// TIA Portal project "Elevador" (V16)

(* hardware
DEVICE "S71500/ET200MP station_1"  S7-1500 station
   slot 0: "Rail_0"  Rack  6ES7 590-1***0-0AA0
   slot 1: "PLC_1"  CPU 1516-3 PN/DP  6ES7 516-3AN00-0AB0  V1.8
      slot 3: "CPU display_1"  6ES7591-1BA00-0AA0
      slot 32768: "PROFINET interface_1"  X1
         slot 32769: "Port_1"  X1 P1
         slot 32770: "Port_2"  X1 P2
      slot 33024: "PROFINET interface_2"  X2
         slot 33025: "Port_1"  X2 P1
      slot 33280: "DP interface_1"  X3
DEVICE "HMI_1"  TP700 Comfort
   slot 0: "HMI_1"  TP700 Comfort  6AV2 124-0GC01-0AX0  16.0.0.0
   slot 1: "HMI_RT_1"  TP700 Comfort  6AV2 124-0GC01-0AX0  16.0.0.0
   slot 5: "HMI_1.IE_CP_1"  PROFINET Interface  16.0.0.0
      slot 1: "PROFINET Interface_1"  PROFINET Interface
         slot 1: "Port_1"  Port
         slot 2: "Port_2"  Port
   slot 7: "HMI_1.MPI/DP_CP_1"  MPI/DP Interface  16.0.0.0
DEVICE "HMI_2"  TP700 Comfort
   slot 0: "HMI_2"  TP700 Comfort  6AV2 124-0GC01-0AX0  16.0.0.0
   slot 1: "HMI_RT_2"  TP700 Comfort  6AV2 124-0GC01-0AX0  16.0.0.0
   slot 5: "HMI_2.IE_CP_1"  PROFINET Interface  16.0.0.0
      slot 1: "PROFINET Interface_1"  PROFINET Interface
         slot 1: "Port_1"  Port
         slot 2: "Port_2"  Port
   slot 7: "HMI_2.MPI/DP_CP_1"  MPI/DP Interface  16.0.0.0
*)

// ===== PLC "PLC_1"  CPU 1516-3 PN/DP =====

VAR_GLOBAL   // PLC tag table "Default tag table"
   "posGround" AT %I0.0 : Bool;   // Sensor Elevador En Planta Baja
   "posFloor1" AT %I0.1 : Bool;   // Sensor Elevador en Primer Piso
   "posFloor2" AT %I0.2 : Bool;   // Sensor Elevador en Segundo Piso
   "posFloor3" AT %I0.3 : Bool;   // Sensor Elevador en Tercer Piso
   "slowGround" AT %I0.4 : Bool;   // Sensor Cambio a Vel Reducida PB
   "slowBottom1" AT %I0.5 : Bool;   // Sensor Cambio Vel Reducida PP Abajo
   "slowTop1" AT %I0.6 : Bool;   // Sensor Cambio Vel Reducida PP Arriba
   "slowBottom2" AT %I0.7 : Bool;   // Sensor Cambio Vel Reducida SP Abajo
   "slowTop2" AT %I1.0 : Bool;   // Sensor Cambio Vel Reducida SP Arriba
   "slow3" AT %I1.1 : Bool;   // Sensor Cambio a Vel Reducida TP
   "doorOpenedG" AT %I1.2 : Bool;   // Sensor Puerta Abierta en Planta Baja
   "doorClosedG" AT %I1.3 : Bool;   // Sensor Puerta Cerrada en Planta Baja
   "doorOpened1" AT %I1.4 : Bool;   // Sensor Puerta Abierta en Primer Piso
   "doorClosed1" AT %I1.5 : Bool;   // Sensor Puerta Cerrada en Primer Piso
   "doorOpened2" AT %I1.6 : Bool;   // Sensor Puerta Abierta en Segundo Piso
   "doorClosed2" AT %I1.7 : Bool;   // Sensor Puerta Cerrada en Segundo Piso
   "doorOpened3" AT %I2.0 : Bool;   // Sensor Puerta Abierta en Tercer Piso
   "doorClosed3" AT %I2.1 : Bool;   // Sensor Puerta Cerrada en Tercer Piso
   "lightBGround" AT %I2.2 : Bool;   // Sensor Luz Puerta en Planta Baja
   "lightB1" AT %I2.3 : Bool;   // Sensor Luz Puerta en Primer Piso
   "lightB2" AT %I2.4 : Bool;   // Sensor Luz Puerta en Segundo Piso
   "lightB3" AT %I2.5 : Bool;   // Sensor Luz Puerta en Tercer Piso
   "sendGround" AT %I4.0 : Bool;   // Boton (NC) para envio a Planta Baja
   "send1" AT %I4.1 : Bool;   // Boton (NC) para envio a Primer Piso
   "send2" AT %I4.2 : Bool;   // Boton (NC) para envio a Segundo Piso
   "send3" AT %I4.3 : Bool;   // Boton (NC) para envio a Tercer Piso
   "alert" AT %I4.4 : Bool;   // Boton (NC) para Alerta
   "emergency" AT %I4.5 : Bool;   // Boton (NC) para Paro Emergencia
   "callGround" AT %I5.0 : Bool;   // Boton (NC) para llamar en Planta Baja
   "callDown1" AT %I5.1 : Bool;   // Boton (NC) para llamar Abajo Primer Piso
   "callUp1" AT %I5.2 : Bool;   // Boton (NC) para llamar Arriba Primer Piso
   "callDown2" AT %I5.3 : Bool;   // Boton (NC) para llamar Abajo Segundo Piso
   "callUp2" AT %I5.4 : Bool;   // Boton (NC) para llamar Arriba Segundo Piso
   "call3" AT %I5.5 : Bool;   // Boton (NC) para llamar en Tercer Piso
   "overload" AT %I5.6 : Bool;   // Boton (NC) de Sobrecarga por Peso
   "toZ+" AT %Q0.0 : Bool;   // Motor Elevador Hacia Arriba
   "toZ-" AT %Q0.1 : Bool;   // Motor Elevador Hacia Abajo
   "slow" AT %Q0.2 : Bool;   // Activar Velocidad Reducida Relevador
   "openDoorG" AT %Q0.3 : Bool;   // Puerta Abrir Planta Baja Piston
   "closeDoorG" AT %Q0.4 : Bool;   // Puerta Cerrar Planta Baja Piston
   "openDoor1" AT %Q0.5 : Bool;   // Puerta Abrir Primer Piso Piston
   "closeDoor1" AT %Q0.6 : Bool;   // Puerta Cerrar Primer Piso Piston
   "openDoor2" AT %Q0.7 : Bool;   // Puerta Abrir Segundo Piso Piston
   "closeDoor2" AT %Q1.0 : Bool;   // Puerta Cerrar Segundo Piso Piston
   "openDoor3" AT %Q1.1 : Bool;   // Puerta Abrir Tercer Piso Piston
   "closeDoor3" AT %Q1.2 : Bool;   // Puerta Cerrar Tercer Piso Piston
   "callToGround" AT %Q1.3 : Bool;   // LED Llamar Planta Baja
   "callToDown1" AT %Q1.4 : Bool;   // LED Llamar Abajo Primer Piso
   "callToUp1" AT %Q1.5 : Bool;   // LED Llamar Arriba Primer Piso
   "callToDown2" AT %Q1.6 : Bool;   // LED Llamar Abajo Segundo Piso
   "callToUp2" AT %Q1.7 : Bool;   // LED Llamar Arriba Segundo Piso
   "callTo3" AT %Q2.0 : Bool;   // LED Llamar Tercer Piso
   "floorIndicatorG" AT %Q2.1 : Bool;   // LED Elevador en Planta Baja
   "floorIndicator1" AT %Q2.2 : Bool;   // LED Elevador en Primer Piso
   "floorIndicator2" AT %Q2.3 : Bool;   // LED Elevador en Segundo Piso
   "floorIndicator3" AT %Q2.4 : Bool;   // LED Elevador en Tercer Piso
   "cabinDown" AT %Q2.5 : Bool;   // LED Elevador Moviendose hacia Abajo
   "cabinUp" AT %Q2.6 : Bool;   // LED Elevador Moviendose hacia Arriba
   "sendToGround" AT %Q2.7 : Bool;   // LED Envio a Planta Baja
   "sendTo1" AT %Q3.0 : Bool;   // LED Envio a Primer Piso
   "sendTo2" AT %Q3.1 : Bool;   // LED Envio a Segundo Piso
   "sendTo3" AT %Q3.2 : Bool;   // LED Envio a Tercer Piso
   "alertInd" AT %Q3.3 : Bool;   // LED Alerta Activada
   "emergencyInd" AT %Q3.4 : Bool;   // LED Paro de Emergencia Activado
   "overloadInd" AT %Q3.5 : Bool;   // LED Sobrecarga Detectada
   "sendGroundMaster" AT %M0.1 : Bool;
   "send1Master" AT %M0.2 : Bool;
   "send2Master" AT %M0.3 : Bool;
   "send3Master" AT %M0.4 : Bool;
   "alertMaster" AT %M0.5 : Bool;
   "emergencyMaster" AT %M0.6 : Bool;
   "abrirPuertasMaster" AT %M0.7 : Bool;
   "cerrarPuertasMaster" AT %M1.0 : Bool;
   "tempFloor1" AT %M1.1 : Bool;
   "tempFloor2" AT %M1.2 : Bool;
   "tempFloor3" AT %M1.3 : Bool;
   "tempFloor4" AT %M1.4 : Bool;
   "tempFloor5" AT %M1.5 : Bool;
   "tempFloor6" AT %M1.6 : Bool;
   "tempFloor7" AT %M1.7 : Bool;
   "sendTo3Master" AT %M2.0 : Bool;
   "sendTo2Master" AT %M2.1 : Bool;
   "sendTo1Master" AT %M2.2 : Bool;
   "sendToGroundMaster" AT %M2.3 : Bool;
   "alertIndMaster" AT %M2.4 : Bool;
   "emergencyIndMaster" AT %M2.5 : Bool;
END_VAR

DATA_BLOCK "Var"   // DB1
{ S7_Optimized_Access := 'TRUE' }
VERSION : 0.1
   VAR
      Acc : Array[0..10] of String;
      AccMovTemp : Array[0..10] of String;
      Ind : Array[0..15] of Bool;
      AccSucc : Array[0..15] of Bool;
      bounceOneAlerta : Bool;
      bounceTwoAlerta : Bool;
      bounceOneEmergen : Bool;
      bounceTwoEmergen : Bool;
      bounceOneGroundA : Bool;
      sendAccGroundA : Bool;
      PuertaIniciada : Bool;
      PuertaAbriendo : Bool;
      PuertaAbierta : Bool;
      PuertaCerrando : Bool;
      PuertaInterrumpida : Bool;
      PuertaTerminada : Bool;
      PuertaTimerInicio : Bool;
      PuertaTimerTermino : Bool;
      PuertaInterrBounce : Bool;
      ActivarPuertaGA : Bool;
      ActivarPuertaF1 : Bool;
      ActivarPuertaF2 : Bool;
      ActivarPuertaF3 : Bool;
      bounceOneF1DownA : Bool;
      sendAccF1DownA : Bool;
      tempStringOne : String;
      tempStringTwo : String;
      ACCION : Bool;
      DeGAaF1 : Bool;
      DeGAaF2 : Bool;
      DeGAaF3 : Bool;
      DeF1aGA : Bool;
      DeF1aF2 : Bool;
      DeF1aF3 : Bool;
      DeF2aGA : Bool;
      DeF2aF1 : Bool;
      DeF2aF3 : Bool;
      DeF3aGA : Bool;
      DeF3aF1 : Bool;
      DeF3aF2 : Bool;
      MOVIMIENTO : Bool;
      MovimientoLento : Bool;
      MovimientoRapido : Bool;
      MASTER : Bool;
      SimuladorEstado1 : Bool;
      SimuladorEstado2 : Bool;
      SimuladorEstado3 : Bool;
      SimuladorEstado4 : Bool;
      SimuladorEstado5 : Bool;
      SimuladorEstado6 : Bool;
      SimuladorEstado7 : Bool;
      SimuladorEstado8 : Bool;
      MASTERINDICATOR : Bool;
      MasterBounceOne : Bool;
      MasterBounceTwo : Bool;
      MasterBounceThree : Bool;
      RESET : Bool;
      ResetApplied : Bool;
      MasterResetPos : Bool;
      MasterResPosPuerta : Bool;
      MasterPuertaG : Bool;
      MasterPuerta1 : Bool;
      MasterPuerta2 : Bool;
      MasterPuerta3 : Bool;
      MasterPuertaGBounce : Bool;
      MasterPuertaGBounce2 : Bool;
      MasterPuerta1Bounce : Bool;
      MasterPuerta1Bounce2 : Bool;
      MasterPuerta2Bounce : Bool;
      MasterPuerta2Bounce2 : Bool;
      MasterPuerta3Bounce : Bool;
      MasterPuerta3Bounce2 : Bool;
      MasterSendToGround : Bool;
      MasterSendTo1 : Bool;
      MasterSendTo2 : Bool;
      MasterSendTo3 : Bool;
      MasterSendToGroundB : Bool;
      MasterSendToGroundB2 : Bool;
      MasterSendTo1B : Bool;
      MasterSendTo1B2 : Bool;
      MasterSendTo2B : Bool;
      MasterSendTo2B2 : Bool;
      MasterSendTo3B : Bool;
      MasterSendTo3B2 : Bool;
      MasterAlertaB1 : Bool;
      MasterAlertaB2 : Bool;
      MasterAlertaB3 : Bool;
      MasterEmergencyB1 : Bool;
      MasterEmergencyB2 : Bool;
      MasterEmergencyB3 : Bool;
      bounceOneF1UpA : Bool;
      sendAccF1UpA : Bool;
      bounceOneF2DownA : Bool;
      sendAccF2DownA : Bool;
      bounceOneF2UpA : Bool;
      sendAccF2UpA : Bool;
      bounceOneF3A : Bool;
      sendAccF3A : Bool;
      bounceGroundPanel : Bool;
      sendAccGroundPanel : Bool;
      bounceF1Panel : Bool;
      sendAccF1Panel : Bool;
      bounceF2Panel : Bool;
      sendAccF2Panel : Bool;
      bounceF3Panel : Bool;
      sendAccF3Panel : Bool;
      bouncePanelF31 : Bool;
      bouncePanelF32 : Bool;
      bouncePanelF33 : Bool;
      bouncePanelF21 : Bool;
      bouncePanelF22 : Bool;
      bouncePanelF23 : Bool;
      bouncePanelF11 : Bool;
      bouncePanelF12 : Bool;
      bouncePanelF13 : Bool;
      bouncePanelFG1 : Bool;
      bouncePanelFG2 : Bool;
      bouncePanelFG3 : Bool;
      Accion2 : Bool;
      Accion3 : Bool;
      TEST : Bool;
      IndTimerInicio : Bool;
      IndTimerTermino : Bool;
      Ultimo : String;
      LimpiarUltimo : Bool;
   END_VAR
BEGIN
   Acc[0] := 'EMPTY';
   Acc[1] := 'EMPTY';
   Acc[2] := 'EMPTY';
   Acc[3] := 'EMPTY';
   Acc[4] := 'EMPTY';
   Acc[5] := 'EMPTY';
   Acc[6] := 'EMPTY';
   Acc[7] := 'EMPTY';
   Acc[8] := 'EMPTY';
   Acc[9] := 'EMPTY';
   Acc[10] := 'EMPTY';
   AccMovTemp[0] := 'EMPTY';
   AccMovTemp[1] := 'EMPTY';
   AccMovTemp[2] := 'EMPTY';
   AccMovTemp[3] := 'EMPTY';
   AccMovTemp[4] := 'EMPTY';
   AccMovTemp[5] := 'EMPTY';
   AccMovTemp[6] := 'EMPTY';
   AccMovTemp[7] := 'EMPTY';
   AccMovTemp[8] := 'EMPTY';
   AccMovTemp[9] := 'EMPTY';
   AccMovTemp[10] := 'EMPTY';
END_DATA_BLOCK

// folder: System blocks/Program resources

DATA_BLOCK "TimAbrir"   // DB2
{ S7_Optimized_Access := 'TRUE' }
AUTHOR : Simatic
FAMILY : IEC
NAME : IEC_TMR
VERSION : 1.0
// stored: InstanceOfName IEC_TIMER
"IEC_TIMER"
BEGIN
END_DATA_BLOCK

// folder: (top level)

FUNCTION "Borrar" : Void   // FC1, SCL
{ S7_Optimized_Access := 'TRUE' }
VERSION : 0.1
   VAR_TEMP
      i : UInt;
      iTwo : UInt;
   END_VAR
   VAR CONSTANT
      INDSIZE : UInt := 10;
   END_VAR
BEGIN
   "Var".Ultimo := "Var".Acc[0];
   "Var".Acc[0] := 'EMPTY';
   FOR #i := 1 TO #INDSIZE DO
       #iTwo := (#i - 1);
       "Var".tempStringOne := "Var".Acc[#i];
       "Var".Acc[#iTwo] := "Var".tempStringOne;
   END_FOR;
   #iTwo := 0;
   "Var".tempStringOne := '';
END_FUNCTION

FUNCTION "Test" : Void   // FC2, SCL
{ S7_Optimized_Access := 'TRUE' }
VERSION : 0.1
BEGIN
   IF "Var".ActivarPuertaGA = FALSE AND "Var".ActivarPuertaF1 = FALSE AND "Var".ActivarPuertaF2 = FALSE AND "Var".ActivarPuertaF3 = FALSE AND "Var".DeGAaF1 = FALSE AND "Var".DeGAaF2 = FALSE AND "Var".DeGAaF3 = FALSE AND "Var".DeF1aGA = FALSE AND "Var".DeF1aF2 = FALSE AND "Var".DeF1aF3 = FALSE AND "Var".DeF2aGA = FALSE AND "Var".DeF2aF1 = FALSE AND "Var".DeF2aF3 = FALSE AND "Var".DeF3aGA = FALSE AND "Var".DeF3aF1 = FALSE AND "Var".DeF3aF2 = FALSE THEN
       "Var".TEST := TRUE;
   ELSE
       "Var".TEST := FALSE;
   END_IF;
END_FUNCTION

ORGANIZATION_BLOCK "Main"   // OB1, LAD, ProgramCycle
TITLE = "Main Program Sweep (Cycle)"
{ S7_Optimized_Access := 'TRUE' }
VERSION : 0.1
   VAR_INPUT
      Initial_Call : Bool;   // Initial call of this OB
      Remanence : Bool;   // =True, if remanent data are available
   END_VAR
   VAR_TEMP
      i : UInt;
      AbrirPuertaTemp : Bool;
      MedPuertaG : Bool;
      iTwo : UInt;
   END_VAR
   VAR CONSTANT
      "TIMER" : Time := T#2S;
      INDSIZE : UInt := 10;
      INDSIZEMOV : UInt := 9;
      EMPTYSTR : UInt := 5;
      TIMERTWO : Time := T#1000ms;
   END_VAR
BEGIN

REGION Network 1 (SCL)
   (*

   20%   Se van guardando en memoria los llamados, es decir que si hay un llamado contrario al actual lo ignorara y lo atendera mas tarde.
   15%        Se puede interrumpir al elevador mientras se mueve siempre y cuando tenga suficiente tiempo para detenerse y recoger a la persona. (SOlo hace caso a los llamados que correspondan al actual.)
   15%  LISTOmmm      El elevador varia de velocidad al acercarse a los pisos adecuados mientras sube o baja.
   10%  LISTO      Existe un HMI simulando las puiertas del elevador y otro con el panel interno del elevador.
   10%  LISTO      En el HMI del panel existe un modo maestro que detiene al elevador y hace control manual mediante el panel, incluyendo abrir y cerrar las puertas. Saliendo del modo manual al automatico reiniciamos al elevador en algun punto. 
   5%   LISTO     El elevador sube y baja correctamente sin salirse de los limites respondiendo a los llamados.
   5%   LISTO     El elevador cierra y abre las puertas correctamente al llegar a los pisos.
   5%   LISTO     Si las puertas en cualquier momento abiertas detectan obstruccion se vuelven a abrir.
   5%   LISTO  La alarma unicamente se activa, el paro detiene todo proceso del elevador.
   5%   LISTO  Si existe sobrepeso con las puertas abiertas entonces no  se cierran y se detiene toda accion, cierran hasta que se quite estado.
   5%   LISTO     Todos los indicadores fueron implementados.
   B Cuando en master no ha llegado a un nivel y cambia direccion

   *)
END_REGION

REGION Network 2 (SCL): Indicadores Basicos
   //IF #Initial_Call = TRUE THEN FILL_BLK(IN := FALSE, COUNT := #INDSIZE, OUT => "Var".Ind[0]); END_IF;

   //LISTO Indicar posicion del elevador si pasa por ese lugar.
   IF "posGround" = TRUE THEN
       "floorIndicatorG" := TRUE;
       "floorIndicator1" := FALSE;
       "floorIndicator2" := FALSE;
       "floorIndicator3" := FALSE;
       "tempFloor1" := TRUE;
       "tempFloor2" := FALSE;
       "tempFloor3" := FALSE;
       "tempFloor4" := FALSE;
       "tempFloor5" := FALSE;
       "tempFloor6" := FALSE;
       "tempFloor7" := FALSE;
   END_IF;

   IF "posFloor3" = TRUE THEN
       "floorIndicatorG" := FALSE;
       "floorIndicator1" := FALSE;
       "floorIndicator2" := FALSE;
       "floorIndicator3" := TRUE;
       "tempFloor1" := FALSE;
       "tempFloor2" := FALSE;
       "tempFloor3" := FALSE;
       "tempFloor4" := FALSE;
       "tempFloor5" := FALSE;
       "tempFloor6" := TRUE;
       "tempFloor7" := FALSE;
   END_IF;

   IF "posFloor1" = TRUE THEN
       IF "tempFloor1" = TRUE THEN
           "floorIndicatorG" := FALSE;
           "floorIndicator1" := TRUE;
           "floorIndicator2" := FALSE;
           "floorIndicator3" := FALSE;
           "tempFloor1" := FALSE;
           "tempFloor2" := TRUE;
           "tempFloor3" := FALSE;
           "tempFloor4" := FALSE;
           "tempFloor5" := FALSE;
           "tempFloor6" := FALSE;
           "tempFloor7" := FALSE;
       ELSIF "tempFloor5" = TRUE OR "tempFloor7" = TRUE THEN
           "floorIndicatorG" := FALSE;
           "floorIndicator1" := TRUE;
           "floorIndicator2" := FALSE;
           "floorIndicator3" := FALSE;
           "tempFloor1" := FALSE;
           "tempFloor2" := FALSE;
           "tempFloor3" := FALSE;
           "tempFloor4" := TRUE;
           "tempFloor5" := FALSE;
           "tempFloor6" := FALSE;
           "tempFloor7" := FALSE;
       END_IF;
   END_IF;

   IF "posFloor2" = TRUE THEN
       IF "tempFloor6" = TRUE THEN
           "floorIndicatorG" := FALSE;
           "floorIndicator1" := FALSE;
           "floorIndicator2" := TRUE;
           "floorIndicator3" := FALSE;
           "tempFloor1" := FALSE;
           "tempFloor2" := FALSE;
           "tempFloor3" := FALSE;
           "tempFloor4" := FALSE;
           "tempFloor5" := FALSE;
           "tempFloor6" := FALSE;
           "tempFloor7" := TRUE;
       ELSIF "tempFloor2" = TRUE OR "tempFloor4" = TRUE THEN
           "floorIndicatorG" := FALSE;
           "floorIndicator1" := FALSE;
           "floorIndicator2" := TRUE;
           "floorIndicator3" := FALSE;
           "tempFloor1" := FALSE;
           "tempFloor2" := FALSE;
           "tempFloor3" := FALSE;
           "tempFloor4" := FALSE;
           "tempFloor5" := TRUE;
           "tempFloor6" := FALSE;
           "tempFloor7" := FALSE;
       END_IF;
   END_IF;


   IF "toZ+" = TRUE THEN
       "cabinUp" := TRUE;
   ELSE
       "cabinUp" := FALSE;
   END_IF;
   IF "toZ-" = TRUE THEN
       "cabinDown" := TRUE;

   ELSE
       "cabinDown" := FALSE;
   END_IF;
   IF "overload" = TRUE THEN
       "overloadInd" := TRUE;
       RESET_TIMER("TimAbrir");
   ELSE
       "overloadInd" := FALSE;
   END_IF;

   //LISTO Indicador de Alarma y Emergencia
   //Cuando ambas estan prendidas

   IF "Var".MASTERINDICATOR = FALSE THEN

       IF "Var".Ind[0] = FALSE AND "alert" = FALSE AND "Var".bounceOneAlerta = FALSE AND "Var".bounceTwoAlerta = FALSE THEN
           "alertInd" := FALSE;
           "alertIndMaster" := FALSE;
       END_IF;
       IF "alertInd" = FALSE AND "Var".bounceOneAlerta = FALSE AND "Var".bounceTwoAlerta = FALSE THEN
           IF "alert" = TRUE THEN
               "Var".Ind[0] := TRUE;
               "Var".bounceOneAlerta := TRUE;
               "Var".MasterAlertaB1 := TRUE;
           END_IF;
           IF "alertMaster" = TRUE THEN
               "Var".Ind[0] := TRUE;
               "Var".bounceOneAlerta := TRUE;
               "Var".MasterAlertaB2 := TRUE;
           END_IF;
       END_IF;
       IF "Var".Ind[0] = TRUE AND "Var".bounceOneAlerta = TRUE THEN
           IF "Var".MasterAlertaB1 = TRUE AND "alert" = FALSE THEN
               "alertInd" := TRUE;
               "alertIndMaster" := TRUE;
               "Var".bounceTwoAlerta := TRUE;
               "Var".MasterAlertaB1 := FALSE;
           END_IF;
           IF "Var".MasterAlertaB2 = TRUE AND "alertMaster" = FALSE THEN
               "alertInd" := TRUE;
               "alertIndMaster" := TRUE;
               "Var".bounceTwoAlerta := TRUE;
               "Var".MasterAlertaB2 := FALSE;
           END_IF;
       END_IF;
       IF "Var".Ind[0] = TRUE AND "Var".bounceOneAlerta = TRUE AND "Var".bounceTwoAlerta = TRUE THEN
           IF "alert" = TRUE THEN
               "Var".Ind[0] := FALSE;
               "Var".MasterAlertaB1 := TRUE;
           END_IF;
           IF "alertMaster" = TRUE THEN
               "Var".Ind[0] := FALSE;
               "Var".MasterAlertaB2 := TRUE;
           END_IF;
       END_IF;
       IF "Var".Ind[0] = FALSE AND "Var".bounceOneAlerta = TRUE AND "Var".bounceTwoAlerta = TRUE THEN
           IF "Var".MasterAlertaB1 = TRUE AND "alert" = FALSE THEN
               "alertInd" := FALSE;
               "alertIndMaster" := FALSE;
               "Var".bounceOneAlerta := FALSE;
               "Var".bounceTwoAlerta := FALSE;
               "Var".MasterAlertaB1 := FALSE;
           END_IF;
           IF "Var".MasterAlertaB2 = TRUE AND "alertMaster" = FALSE THEN
               "alertInd" := FALSE;
               "alertIndMaster" := FALSE;
               "Var".bounceOneAlerta := FALSE;
               "Var".bounceTwoAlerta := FALSE;
               "Var".MasterAlertaB2 := FALSE;
           END_IF;
       END_IF;

       IF "Var".Ind[1] = FALSE AND "emergency" = FALSE AND "Var".bounceOneEmergen = FALSE AND "Var".bounceTwoEmergen = FALSE THEN
           "emergencyInd" := FALSE;
           "emergencyIndMaster" := FALSE;
       END_IF;
       IF "emergencyInd" = FALSE AND "Var".bounceOneEmergen = FALSE AND "Var".bounceTwoEmergen = FALSE THEN
           IF "emergency" = TRUE THEN
               "Var".Ind[1] := TRUE;
               "Var".bounceOneEmergen := TRUE;
               "Var".MasterEmergencyB1 := TRUE;
           END_IF;
           IF "emergencyMaster" = TRUE THEN
               "Var".Ind[1] := TRUE;
               "Var".bounceOneEmergen := TRUE;
               "Var".MasterEmergencyB2 := TRUE;
           END_IF;
       END_IF;
       IF "Var".Ind[1] = TRUE AND "Var".bounceOneEmergen = TRUE THEN
           IF "Var".MasterEmergencyB1 = TRUE AND "emergency" = FALSE THEN
               "emergencyInd" := TRUE;
               "emergencyIndMaster" := TRUE;
               "Var".bounceTwoEmergen := TRUE;
               "Var".MasterEmergencyB1 := FALSE;
           END_IF;
           IF "Var".MasterEmergencyB2 = TRUE AND "emergencyMaster" = FALSE THEN
               "emergencyInd" := TRUE;
               "emergencyIndMaster" := TRUE;
               "Var".bounceTwoEmergen := TRUE;
               "Var".MasterEmergencyB2 := FALSE;
           END_IF;
       END_IF;
       IF "Var".Ind[1] = TRUE AND "Var".bounceOneEmergen = TRUE AND "Var".bounceTwoEmergen = TRUE THEN
           IF "emergency" = TRUE THEN
               "Var".Ind[1] := FALSE;
               "Var".MasterEmergencyB1 := TRUE;
           END_IF;
           IF "emergencyMaster" = TRUE THEN
               "Var".Ind[1] := FALSE;
               "Var".MasterEmergencyB2 := TRUE;
           END_IF;
       END_IF;
       IF "Var".Ind[1] = FALSE AND "Var".bounceOneEmergen = TRUE AND "Var".bounceTwoEmergen = TRUE THEN
           IF "Var".MasterEmergencyB1 = TRUE AND "emergency" = FALSE THEN
               "emergencyInd" := FALSE;
               "emergencyIndMaster" := FALSE;
               "Var".bounceOneEmergen := FALSE;
               "Var".bounceTwoEmergen := FALSE;
               "Var".MasterEmergencyB1 := FALSE;
               "Var".ResetApplied := FALSE;
               "Var".MasterResetPos := TRUE;
           END_IF;
           IF "Var".MasterEmergencyB2 = TRUE AND "emergencyMaster" = FALSE THEN
               "emergencyInd" := FALSE;
               "emergencyIndMaster" := FALSE;
               "Var".bounceOneEmergen := FALSE;
               "Var".bounceTwoEmergen := FALSE;
               "Var".MasterEmergencyB2 := FALSE;
               "Var".ResetApplied := FALSE;
               "Var".MasterResetPos := TRUE;
           END_IF;
       END_IF;

   END_IF;

   IF ("emergencyInd" = TRUE OR "emergencyIndMaster" = TRUE) THEN
       IF "Var".ResetApplied = FALSE THEN
           "Var".RESET := TRUE;
           "Var".ResetApplied := TRUE;
       END_IF;
   END_IF;

   IF "Var".MASTERINDICATOR = TRUE THEN
       IF "Var".ResetApplied = FALSE THEN
           "Var".RESET := TRUE;
           "Var".ResetApplied := TRUE;
       END_IF;
   END_IF;
END_REGION

REGION Network 3 (SCL): Agregar Acciones Lista
   IF "Var".MASTERINDICATOR = FALSE THEN

       //Notar que los indicadore de array se quedan encendidos hasta acabar accion de la puerta
       //GA, F1DA, F1UA, F2DA, F2UA, F3A, GFP, F1P, F2P, F3P

       REGION AgregarCallGroundAfuera
           IF "Var".Ind[2] = FALSE AND "callGround" = FALSE AND "Var".bounceOneGroundA = FALSE THEN "callToGround" := FALSE; END_IF;
           IF "callToGround" = FALSE AND "callGround" = TRUE AND "Var".bounceOneGroundA = FALSE THEN "Var".Ind[2] := TRUE; "Var".bounceOneGroundA := TRUE; END_IF;
           IF "Var".Ind[2] = TRUE AND "callGround" = FALSE AND "Var".bounceOneGroundA = TRUE THEN "callToGround" := TRUE; "Var".bounceOneGroundA := FALSE; "Var".sendAccGroundA := TRUE; END_IF;
           IF "Var".Ind[2] = TRUE AND "Var".sendAccGroundA = TRUE AND "Var".AccSucc[2] = FALSE THEN
               FOR #i := 0 TO #INDSIZE DO
                   IF LEN("Var".Acc[#i]) = #EMPTYSTR AND "Var".AccSucc[2] = FALSE THEN
                       "Var".Acc[#i] := 'GA';
                       "Var".AccSucc[2] := TRUE;
                   END_IF;
               END_FOR;
               "Var".sendAccGroundA := FALSE;
               "Var".AccSucc[2] := FALSE;
           END_IF;
       END_REGION ;

       REGION AgregarCallF1Abajo
           IF "Var".Ind[3] = FALSE AND "callDown1" = FALSE AND "Var".bounceOneF1DownA = FALSE THEN "callToDown1" := FALSE; END_IF;
           IF "callToDown1" = FALSE AND "callDown1" = TRUE AND "Var".Ind[3] = FALSE AND "Var".bounceOneF1DownA = FALSE THEN "Var".Ind[3] := TRUE; "Var".bounceOneF1DownA := TRUE; END_IF;
           IF "Var".Ind[3] = TRUE AND "callDown1" = FALSE AND "Var".bounceOneF1DownA = TRUE THEN "callToDown1" := TRUE; "Var".bounceOneF1DownA := FALSE; "Var".sendAccF1DownA := TRUE; END_IF;
           IF "Var".Ind[3] = TRUE AND "Var".sendAccF1DownA = TRUE AND "Var".AccSucc[3] = FALSE THEN
               FOR #i := 0 TO #INDSIZE DO
                   IF LEN("Var".Acc[#i]) = #EMPTYSTR AND "Var".AccSucc[3] = FALSE THEN
                       "Var".Acc[#i] := 'F1DA';
                       "Var".AccSucc[3] := TRUE;
                   END_IF;
               END_FOR;
               "Var".sendAccF1DownA := FALSE;
               "Var".AccSucc[3] := FALSE;
           END_IF;
       END_REGION ;

       REGION AgregarCallF1Arriba
           IF "Var".Ind[4] = FALSE AND "callUp1" = FALSE AND "Var".bounceOneF1UpA = FALSE THEN "callToUp1" := FALSE; END_IF;
           IF "callToUp1" = FALSE AND "callUp1" = TRUE AND "Var".Ind[4] = FALSE AND "Var".bounceOneF1UpA = FALSE THEN "Var".Ind[4] := TRUE; "Var".bounceOneF1UpA := TRUE; END_IF;
           IF "Var".Ind[4] = TRUE AND "callUp1" = FALSE AND "Var".bounceOneF1UpA = TRUE THEN "callToUp1" := TRUE; "Var".bounceOneF1UpA := FALSE; "Var".sendAccF1UpA := TRUE; END_IF;
           IF "Var".Ind[4] = TRUE AND "Var".sendAccF1UpA = TRUE AND "Var".AccSucc[4] = FALSE THEN
               FOR #i := 0 TO #INDSIZE DO
                   IF LEN("Var".Acc[#i]) = #EMPTYSTR AND "Var".AccSucc[4] = FALSE THEN
                       "Var".Acc[#i] := 'F1UA';
                       "Var".AccSucc[4] := TRUE;
                   END_IF;
               END_FOR;
               "Var".sendAccF1UpA := FALSE;
               "Var".AccSucc[4] := FALSE;
           END_IF;
       END_REGION ;

       REGION AgregarCallF2Abajo
           IF "Var".Ind[5] = FALSE AND "callDown2" = FALSE AND "Var".bounceOneF2DownA = FALSE THEN "callToDown2" := FALSE; END_IF;
           IF "callToDown2" = FALSE AND "callDown2" = TRUE AND "Var".Ind[5] = FALSE AND "Var".bounceOneF2DownA = FALSE THEN "Var".Ind[5] := TRUE; "Var".bounceOneF2DownA := TRUE; END_IF;
           IF "Var".Ind[5] = TRUE AND "callDown2" = FALSE AND "Var".bounceOneF2DownA = TRUE THEN "callToDown2" := TRUE; "Var".bounceOneF2DownA := FALSE; "Var".sendAccF2DownA := TRUE; END_IF;
           IF "Var".Ind[5] = TRUE AND "Var".sendAccF2DownA = TRUE AND "Var".AccSucc[5] = FALSE THEN
               FOR #i := 0 TO #INDSIZE DO
                   IF LEN("Var".Acc[#i]) = #EMPTYSTR AND "Var".AccSucc[5] = FALSE THEN
                       "Var".Acc[#i] := 'F2DA';
                       "Var".AccSucc[5] := TRUE;
                   END_IF;
               END_FOR;
               "Var".sendAccF2DownA := FALSE;
               "Var".AccSucc[5] := FALSE;
           END_IF;
       END_REGION ;

       REGION AgregarCallF2Arriba
           IF "Var".Ind[6] = FALSE AND "callUp2" = FALSE AND "Var".bounceOneF2UpA = FALSE THEN "callToUp2" := FALSE; END_IF;
           IF "callToUp2" = FALSE AND "callUp2" = TRUE  AND "Var".Ind[6] = FALSE AND "Var".bounceOneF2UpA = FALSE THEN "Var".Ind[6] := TRUE; "Var".bounceOneF2UpA := TRUE; END_IF;
           IF "Var".Ind[6] = TRUE AND "callUp2" = FALSE AND "Var".bounceOneF2UpA = TRUE THEN "callToUp2" := TRUE; "Var".bounceOneF2UpA := FALSE; "Var".sendAccF2UpA := TRUE; END_IF;
           IF "Var".Ind[6] = TRUE AND "Var".sendAccF2UpA = TRUE AND "Var".AccSucc[6] = FALSE THEN
               FOR #i := 0 TO #INDSIZE DO
                   IF LEN("Var".Acc[#i]) = #EMPTYSTR AND "Var".AccSucc[6] = FALSE THEN
                       "Var".Acc[#i] := 'F2UA';
                       "Var".AccSucc[6] := TRUE;
                   END_IF;
               END_FOR;
               "Var".sendAccF2UpA := FALSE;
               "Var".AccSucc[6] := FALSE;
           END_IF;
       END_REGION ;

       REGION AgregarCallF3Afuera 
           IF "Var".Ind[7] = FALSE AND "call3" = FALSE AND "Var".bounceOneF3A = FALSE THEN "callTo3" := FALSE; END_IF;
           IF "callTo3" = FALSE AND "call3" = TRUE AND "Var".bounceOneF3A = FALSE THEN "Var".Ind[7] := TRUE; "Var".bounceOneF3A := TRUE; END_IF;
           IF "Var".Ind[7] = TRUE AND "call3" = FALSE AND "Var".bounceOneF3A = TRUE THEN "callTo3" := TRUE; "Var".bounceOneF3A := FALSE; "Var".sendAccF3A := TRUE; END_IF;
           IF "Var".Ind[7] = TRUE AND "Var".sendAccF3A = TRUE AND "Var".AccSucc[7] = FALSE THEN
               FOR #i := 0 TO #INDSIZE DO
                   IF LEN("Var".Acc[#i]) = #EMPTYSTR AND "Var".AccSucc[7] = FALSE THEN
                       "Var".Acc[#i] := 'F3A';
                       "Var".AccSucc[7] := TRUE;
                   END_IF;
               END_FOR;
               "Var".sendAccF3A := FALSE;
               "Var".AccSucc[7] := FALSE;
           END_IF;
       END_REGION;


       REGION AgregarCallPanelG
           IF "Var".Ind[8] = FALSE AND "sendGround" = FALSE AND "Var".bouncePanelFG1 = FALSE THEN
               "sendToGround" := FALSE;
               "sendToGroundMaster" := FALSE;
           END_IF;
           IF "sendToGround" = FALSE AND "Var".bouncePanelFG1 = FALSE THEN
               IF "sendGround" = TRUE THEN
                   "Var".Ind[8] := TRUE;
                   "Var".bouncePanelFG1 := TRUE;
                   "Var".bouncePanelFG2 := TRUE;
               END_IF;
               IF "sendGroundMaster" = TRUE THEN
                   "Var".Ind[8] := TRUE;
                   "Var".bouncePanelFG1 := TRUE;
                   "Var".bouncePanelFG3 := TRUE;
               END_IF;
           END_IF;
           IF "Var".Ind[8] = TRUE AND "Var".bouncePanelFG1 = TRUE THEN
               IF "Var".bouncePanelFG2 = TRUE AND "sendGround" = FALSE THEN
                   "sendToGround" := TRUE;
                   "sendToGroundMaster" := TRUE;
                   "Var".bouncePanelFG1 := FALSE;
                   "Var".bouncePanelFG2 := FALSE;
                   "Var".sendAccGroundPanel := TRUE;
               END_IF;
               IF "Var".bouncePanelFG3 = TRUE AND "sendGroundMaster" = FALSE THEN
                   "sendToGround" := TRUE;
                   "sendToGroundMaster" := TRUE;
                   "Var".bouncePanelFG1 := FALSE;
                   "Var".bouncePanelFG3 := FALSE;
                   "Var".sendAccGroundPanel := TRUE;
               END_IF;
           END_IF;
           IF "Var".Ind[8] = TRUE AND "Var".sendAccGroundPanel = TRUE AND "Var".AccSucc[8] = FALSE THEN
               FOR #i := 0 TO #INDSIZE DO
                   IF LEN("Var".Acc[#i]) = #EMPTYSTR AND "Var".AccSucc[8] = FALSE THEN
                       "Var".Acc[#i] := 'GFP';
                       "Var".AccSucc[8] := TRUE;
                   END_IF;
               END_FOR;
               "Var".sendAccGroundPanel := FALSE;
               "Var".AccSucc[8] := FALSE;
           END_IF;
       END_REGION ;

       REGION AgregarCallPanelF1
           IF "Var".Ind[9] = FALSE AND "send1" = FALSE AND "Var".bouncePanelF11 = FALSE THEN
               "sendTo1" := FALSE;
               "sendTo1Master" := FALSE;
           END_IF;
           IF "sendTo1" = FALSE AND "Var".bouncePanelF11 = FALSE THEN
               IF "send1" = TRUE THEN
                   "Var".Ind[9] := TRUE;
                   "Var".bouncePanelF11 := TRUE;
                   "Var".bouncePanelF12 := TRUE;
               END_IF;
               IF "send1Master" = TRUE THEN
                   "Var".Ind[9] := TRUE;
                   "Var".bouncePanelF11 := TRUE;
                   "Var".bouncePanelF13 := TRUE;
               END_IF;
           END_IF;
           IF "Var".Ind[9] = TRUE AND "Var".bouncePanelF11 = TRUE THEN
               IF "Var".bouncePanelF12 = TRUE AND "send1" = FALSE THEN
                   "sendTo1" := TRUE;
                   "sendTo1Master" := TRUE;
                   "Var".bouncePanelF11 := FALSE;
                   "Var".bouncePanelF12 := FALSE;
                   "Var".sendAccF1Panel := TRUE;
               END_IF;
               IF "Var".bouncePanelF13 = TRUE AND "send1Master" = FALSE THEN
                   "sendTo1" := TRUE;
                   "sendTo1Master" := TRUE;
                   "Var".bouncePanelF11 := FALSE;
                   "Var".bouncePanelF13 := FALSE;
                   "Var".sendAccF1Panel := TRUE;
               END_IF;
           END_IF;
           IF "Var".Ind[9] = TRUE AND "Var".sendAccF1Panel = TRUE AND "Var".AccSucc[9] = FALSE THEN
               FOR #i := 0 TO #INDSIZE DO
                   IF LEN("Var".Acc[#i]) = #EMPTYSTR AND "Var".AccSucc[9] = FALSE THEN
                       "Var".Acc[#i] := 'F1P';
                       "Var".AccSucc[9] := TRUE;
                   END_IF;
               END_FOR;
               "Var".sendAccF1Panel := FALSE;
               "Var".AccSucc[9] := FALSE;
           END_IF;
       END_REGION ;

       REGION AgregarCallPanelF2
           IF "Var".Ind[10] = FALSE AND "send2" = FALSE AND "Var".bouncePanelF21 = FALSE THEN
               "sendTo2" := FALSE;
               "sendTo2Master" := FALSE;
           END_IF;
           IF "sendTo2" = FALSE AND "Var".bouncePanelF21 = FALSE THEN
               IF "send2" = TRUE THEN
                   "Var".Ind[10] := TRUE;
                   "Var".bouncePanelF21 := TRUE;
                   "Var".bouncePanelF22 := TRUE;
               END_IF;
               IF "send2Master" = TRUE THEN
                   "Var".Ind[10] := TRUE;
                   "Var".bouncePanelF21 := TRUE;
                   "Var".bouncePanelF23 := TRUE;
               END_IF;
           END_IF;
           IF "Var".Ind[10] = TRUE AND "Var".bouncePanelF21 = TRUE THEN
               IF "Var".bouncePanelF22 = TRUE AND "send2" = FALSE THEN
                   "sendTo2" := TRUE;
                   "sendTo2Master" := TRUE;
                   "Var".bouncePanelF21 := FALSE;
                   "Var".bouncePanelF22 := FALSE;
                   "Var".sendAccF2Panel := TRUE;
               END_IF;
               IF "Var".bouncePanelF23 = TRUE AND "send2Master" = FALSE THEN
                   "sendTo2" := TRUE;
                   "sendTo2Master" := TRUE;
                   "Var".bouncePanelF21 := FALSE;
                   "Var".bouncePanelF23 := FALSE;
                   "Var".sendAccF2Panel := TRUE;
               END_IF;
           END_IF;
           IF "Var".Ind[10] = TRUE AND "Var".sendAccF2Panel = TRUE AND "Var".AccSucc[10] = FALSE THEN
               FOR #i := 0 TO #INDSIZE DO
                   IF LEN("Var".Acc[#i]) = #EMPTYSTR AND "Var".AccSucc[10] = FALSE THEN
                       "Var".Acc[#i] := 'F2P';
                       "Var".AccSucc[10] := TRUE;
                   END_IF;
               END_FOR;
               "Var".sendAccF2Panel := FALSE;
               "Var".AccSucc[10] := FALSE;
           END_IF;
       END_REGION ;

       REGION AgregarCallPanelF3
           IF "Var".Ind[11] = FALSE AND "send3" = FALSE AND "Var".bouncePanelF31 = FALSE THEN "sendTo3" := FALSE; "sendTo3Master" := FALSE; END_IF;
           IF "sendTo3" = FALSE AND "Var".bouncePanelF31 = FALSE THEN
               IF "send3" = TRUE THEN
                   "Var".Ind[11] := TRUE;
                   "Var".bouncePanelF31 := TRUE;
                   "Var".bouncePanelF32 := TRUE;
               END_IF;
               IF "send3Master" = TRUE THEN
                   "Var".Ind[11] := TRUE;
                   "Var".bouncePanelF31 := TRUE;
                   "Var".bouncePanelF33 := TRUE;
               END_IF;
           END_IF;
           IF "Var".Ind[11] = TRUE AND "Var".bouncePanelF31 = TRUE THEN
               IF "Var".bouncePanelF32 = TRUE AND "send3" = FALSE THEN
                   "sendTo3" := TRUE;
                   "sendTo3Master" := TRUE;
                   "Var".bouncePanelF31 := FALSE;
                   "Var".bouncePanelF32 := FALSE;
                   "Var".sendAccF3Panel := TRUE;
               END_IF;
               IF "Var".bouncePanelF33 = TRUE AND "send3Master" = FALSE THEN
                   "sendTo3" := TRUE;
                   "sendTo3Master" := TRUE;
                   "Var".bouncePanelF31 := FALSE;
                   "Var".bouncePanelF33 := FALSE;
                   "Var".sendAccF3Panel := TRUE;
               END_IF;
           END_IF;
           IF "Var".Ind[11] = TRUE AND "Var".sendAccF3Panel = TRUE AND "Var".AccSucc[11] = FALSE THEN
               FOR #i := 0 TO #INDSIZE DO
                   IF LEN("Var".Acc[#i]) = #EMPTYSTR AND "Var".AccSucc[11] = FALSE THEN
                       "Var".Acc[#i] := 'F3P';
                       "Var".AccSucc[11] := TRUE;
                   END_IF;
               END_FOR;
               "Var".sendAccF3Panel := FALSE;
               "Var".AccSucc[11] := FALSE;
           END_IF;
       END_REGION ;



   END_IF;
END_REGION

REGION Network 4 (SCL): ACCIONES
   IF "Var".MASTERINDICATOR = FALSE THEN

       IF "Var".ACCION = FALSE THEN

           REGION AccionesGA
               "Test"();
               IF "Var".Acc[0] = 'GA' AND "posGround" = TRUE AND "Var".TEST = TRUE THEN
                   "Borrar"();
                   "Var".Ind[2] := FALSE;
                   "Var".ActivarPuertaGA := TRUE;
                   "Var".ACCION := TRUE;
               END_IF;
               "Test"();
               IF "Var".Acc[0] = 'GA' AND "posFloor1" = TRUE AND "Var".TEST = TRUE THEN
                   "Borrar"();
                   "Var".DeF1aGA := TRUE;
                   "Var".ACCION := TRUE;
               END_IF;
               "Test"();
               IF "Var".Acc[0] = 'GA' AND "posFloor2" = TRUE AND "Var".TEST = TRUE THEN
                   "Borrar"();
                   "Var".DeF2aGA := TRUE;
                   "Var".ACCION := TRUE;
               END_IF;
               "Test"();
               IF "Var".Acc[0] = 'GA' AND "posFloor3" = TRUE AND "Var".TEST = TRUE THEN
                   "Borrar"();
                   "Var".DeF3aGA := TRUE;
                   "Var".ACCION := TRUE;
               END_IF;
           END_REGION ;

           REGION AccionesF1Down
               "Test"();
               IF "Var".Acc[0] = 'F1DA' AND "posFloor1" = TRUE AND "Var".TEST = TRUE THEN
                   "Borrar"();
                   "Var".Ind[3] := FALSE;
                   "Var".ActivarPuertaF1 := TRUE;
                   "Var".ACCION := TRUE;
               END_IF;
               "Test"();
               IF "Var".Acc[0] = 'F1DA' AND "posGround" = TRUE AND "Var".TEST = TRUE THEN
                   "Borrar"();
                   "Var".DeGAaF1 := TRUE;
                   "Var".ACCION := TRUE;
               END_IF;
               "Test"();
               IF "Var".Acc[0] = 'F1DA' AND "posFloor2" = TRUE AND "Var".TEST = TRUE THEN
                   "Borrar"();
                   "Var".DeF2aF1 := TRUE;
                   "Var".ACCION := TRUE;
               END_IF;
               "Test"();
               IF "Var".Acc[0] = 'F1DA' AND "posFloor3" = TRUE AND "Var".TEST = TRUE THEN
                   "Borrar"();
                   "Var".DeF3aF1 := TRUE;
                   "Var".ACCION := TRUE;
               END_IF;
           END_REGION ;

           REGION AccionesF1Up
               "Test"();
               IF "Var".Acc[0] = 'F1UA' AND "posFloor1" = TRUE AND "Var".TEST = TRUE THEN
                   "Borrar"();
                   "Var".Ind[4] := FALSE;
                   "Var".ActivarPuertaF1 := TRUE;
                   "Var".ACCION := TRUE;
               END_IF;
               "Test"();
               IF "Var".Acc[0] = 'F1UA' AND "posGround" = TRUE AND "Var".TEST = TRUE THEN
                   "Borrar"();
                   "Var".DeGAaF1 := TRUE;
                   "Var".ACCION := TRUE;
               END_IF;
               "Test"();
               IF "Var".Acc[0] = 'F1UA' AND "posFloor2" = TRUE AND "Var".TEST = TRUE THEN
                   "Borrar"();
                   "Var".DeF2aF1 := TRUE;
                   "Var".ACCION := TRUE;
               END_IF;
               "Test"();
               IF "Var".Acc[0] = 'F1UA' AND "posFloor3" = TRUE AND "Var".TEST = TRUE THEN
                   "Borrar"();
                   "Var".DeF3aF1 := TRUE;
                   "Var".ACCION := TRUE;
               END_IF;
           END_REGION ;

           REGION AccionesF2Down
               "Test"();
               IF "Var".Acc[0] = 'F2DA' AND "posFloor2" = TRUE AND "Var".TEST = TRUE THEN
                   "Borrar"();
                   "Var".Ind[5] := FALSE;
                   "Var".ActivarPuertaF2 := TRUE;
                   "Var".ACCION := TRUE;
               END_IF;
               "Test"();
               IF "Var".Acc[0] = 'F2DA' AND "posGround" = TRUE AND "Var".TEST = TRUE THEN
                   "Borrar"();
                   "Var".DeGAaF2 := TRUE;
                   "Var".ACCION := TRUE;
               END_IF;
               "Test"();
               IF "Var".Acc[0] = 'F2DA' AND "posFloor1" = TRUE AND "Var".TEST = TRUE THEN
                   "Borrar"();
                   "Var".DeF1aF2 := TRUE;
                   "Var".ACCION := TRUE;
               END_IF;
               "Test"();
               IF "Var".Acc[0] = 'F2DA' AND "posFloor3" = TRUE AND "Var".TEST = TRUE THEN
                   "Borrar"();
                   "Var".DeF3aF2 := TRUE;
                   "Var".ACCION := TRUE;
               END_IF;
           END_REGION ;

           REGION AccionesF2Up
               "Test"();
               IF "Var".Acc[0] = 'F2UA' AND "posFloor2" = TRUE AND "Var".TEST = TRUE THEN
                   "Borrar"();
                   "Var".Ind[6] := FALSE;
                   "Var".ActivarPuertaF2 := TRUE;
                   "Var".ACCION := TRUE;
               END_IF;
               "Test"();
               IF "Var".Acc[0] = 'F2UA' AND "posGround" = TRUE AND "Var".TEST = TRUE THEN
                   "Borrar"();
                   "Var".DeGAaF2 := TRUE;
                   "Var".ACCION := TRUE;
               END_IF;
               "Test"();
               IF "Var".Acc[0] = 'F2UA' AND "posFloor1" = TRUE AND "Var".TEST = TRUE THEN
                   "Borrar"();
                   "Var".DeF1aF2 := TRUE;
                   "Var".ACCION := TRUE;
               END_IF;
               "Test"();
               IF "Var".Acc[0] = 'F2UA' AND "posFloor3" = TRUE AND "Var".TEST = TRUE THEN
                   "Borrar"();
                   "Var".DeF3aF2 := TRUE;
                   "Var".ACCION := TRUE;
               END_IF;
           END_REGION;

           REGION AccionesF3A
               "Test"();
               IF "Var".Acc[0] = 'F3A' AND "posFloor3" = TRUE AND "Var".TEST = TRUE THEN
                   "Borrar"();
                   "Var".Ind[7] := FALSE;
                   "Var".ActivarPuertaF3 := TRUE;
                   "Var".ACCION := TRUE;
               END_IF;
               "Test"();
               IF "Var".Acc[0] = 'F3A' AND "posGround" = TRUE AND "Var".TEST = TRUE THEN
                   "Borrar"();
                   "Var".DeGAaF3 := TRUE;
                   "Var".ACCION := TRUE;
               END_IF;
               "Test"();
               IF "Var".Acc[0] = 'F3A' AND "posFloor1" = TRUE AND "Var".TEST = TRUE THEN
                   "Borrar"();
                   "Var".DeF1aF3 := TRUE;
                   "Var".ACCION := TRUE;
               END_IF;
               "Test"();
               IF "Var".Acc[0] = 'F3A' AND "posFloor2" = TRUE AND "Var".TEST = TRUE THEN
                   "Borrar"();
                   "Var".DeF2aF3 := TRUE;
                   "Var".ACCION := TRUE;
               END_IF;
           END_REGION ;

           REGION AccionesGFP
               "Test"();
               IF "Var".Acc[0] = 'GFP' AND "posGround" = TRUE AND "Var".TEST = TRUE THEN
                   "Borrar"();
                   "Var".Ind[8] := FALSE;
                   "Var".ActivarPuertaGA := TRUE;
                   "Var".ACCION := TRUE;
               END_IF;
               "Test"();
               IF "Var".Acc[0] = 'GFP' AND "posFloor1" = TRUE AND "Var".TEST = TRUE THEN
                   "Borrar"();
                   "Var".DeF1aGA := TRUE;
                   "Var".ACCION := TRUE;
               END_IF;
               "Test"();
               IF "Var".Acc[0] = 'GFP' AND "posFloor2" = TRUE AND "Var".TEST = TRUE THEN
                   "Borrar"();
                   "Var".DeF2aGA := TRUE;
                   "Var".ACCION := TRUE;
               END_IF;
               "Test"();
               IF "Var".Acc[0] = 'GFP' AND "posFloor3" = TRUE AND "Var".TEST = TRUE THEN
                   "Borrar"();
                   "Var".DeF3aGA := TRUE;
                   "Var".ACCION := TRUE;
               END_IF;
           END_REGION ;

           REGION AccionesF1P
               "Test"();
               IF "Var".Acc[0] = 'F1P' AND "posFloor1" = TRUE AND "Var".TEST = TRUE THEN
                   "Borrar"();
                   "Var".Ind[9] := FALSE;
                   "Var".ActivarPuertaF1 := TRUE;
                   "Var".ACCION := TRUE;
               END_IF;
               "Test"();
               IF "Var".Acc[0] = 'F1P' AND "posGround" = TRUE AND "Var".TEST = TRUE THEN
                   "Borrar"();
                   "Var".DeGAaF1 := TRUE;
                   "Var".ACCION := TRUE;
               END_IF;
               "Test"();
               IF "Var".Acc[0] = 'F1P' AND "posFloor2" = TRUE AND "Var".TEST = TRUE THEN
                   "Borrar"();
                   "Var".DeF2aF1 := TRUE;
                   "Var".ACCION := TRUE;
               END_IF;
               "Test"();
               IF "Var".Acc[0] = 'F1P' AND "posFloor3" = TRUE AND "Var".TEST = TRUE THEN
                   "Borrar"();
                   "Var".DeF3aF1 := TRUE;
                   "Var".ACCION := TRUE;
               END_IF;
           END_REGION ;

           REGION AccionesF2P
               "Test"();
               IF "Var".Acc[0] = 'F2P' AND "posFloor2" = TRUE AND "Var".TEST = TRUE THEN
                   "Borrar"();
                   "Var".Ind[10] := FALSE;
                   "Var".ActivarPuertaF2 := TRUE;
                   "Var".ACCION := TRUE;
               END_IF;
               "Test"();
               IF "Var".Acc[0] = 'F2P' AND "posGround" = TRUE AND "Var".TEST = TRUE THEN
                   "Borrar"();
                   "Var".DeGAaF2 := TRUE;
                   "Var".ACCION := TRUE;
               END_IF;
               "Test"();
               IF "Var".Acc[0] = 'F2P' AND "posFloor1" = TRUE AND "Var".TEST = TRUE THEN
                   "Borrar"();
                   "Var".DeF1aF2 := TRUE;
                   "Var".ACCION := TRUE;
               END_IF;
               "Test"();
               IF "Var".Acc[0] = 'F2P' AND "posFloor3" = TRUE AND "Var".TEST = TRUE THEN
                   "Borrar"();
                   "Var".DeF3aF2 := TRUE;
                   "Var".ACCION := TRUE;
               END_IF;
           END_REGION;

           REGION AccionesF3P
               "Test"();
               IF "Var".Acc[0] = 'F3P' AND "posFloor3" = TRUE AND "Var".TEST = TRUE THEN
                   "Borrar"();
                   "Var".Ind[11] := FALSE;
                   "Var".ActivarPuertaF3 := TRUE;
                   "Var".ACCION := TRUE;
               END_IF;
               "Test"();
               IF "Var".Acc[0] = 'F3P' AND "posGround" = TRUE AND "Var".TEST = TRUE THEN
                   "Borrar"();
                   "Var".DeGAaF3 := TRUE;
                   "Var".ACCION := TRUE;
               END_IF;
               "Test"();
               IF "Var".Acc[0] = 'F3P' AND "posFloor1" = TRUE AND "Var".TEST = TRUE THEN
                   "Borrar"();
                   "Var".DeF1aF3 := TRUE;
                   "Var".ACCION := TRUE;
               END_IF;
               "Test"();
               IF "Var".Acc[0] = 'F3P' AND "posFloor2" = TRUE AND "Var".TEST = TRUE THEN
                   "Borrar"();
                   "Var".DeF2aF3 := TRUE;
                   "Var".ACCION := TRUE;
               END_IF;
           END_REGION ;

           (*
           REGION Validar
               IF "Var".Acc[0] = 'GFP' AND "Var".Ultimo = 'GA' THEN
                   "Var".Acc[0] := 'EMPTY';
                   FOR #i := 1 TO #INDSIZEMOV DO
                       #iTwo := (#i - 1);
                       "Var".tempStringOne := "Var".Acc[#i];
                       "Var".Acc[#iTwo] := "Var".tempStringOne;
                   END_FOR;
                   #iTwo := 0;
                   "Var".tempStringOne := '';
                   "Var".LimpiarUltimo := TRUE;
               END_IF;

               IF "Var".Acc[0] = 'GA' AND "Var".Ultimo = 'GFP' THEN
                   "Var".Acc[0] := 'EMPTY';
                   FOR #i := 1 TO #INDSIZEMOV DO
                       #iTwo := (#i - 1);
                       "Var".tempStringOne := "Var".Acc[#i];
                       "Var".Acc[#iTwo] := "Var".tempStringOne;
                   END_FOR;
                   #iTwo := 0;
                   "Var".tempStringOne := '';
                   "Var".LimpiarUltimo := TRUE;
               END_IF;

               IF "Var".TEST = TRUE AND "Var".IndTimerInicio = FALSE AND "Var".LimpiarUltimo = TRUE THEN
                   "Var".IndTimerInicio := TRUE;
                   "Var".LimpiarUltimo := FALSE;
               END_IF;

               "TimInd".TON(IN := "Var".IndTimerInicio,
                            PT := #TIMERTWO,
                            Q  => "Var".IndTimerTermino);

               IF "Var".IndTimerTermino = TRUE THEN
                   RESET_TIMER("TimInd");
                   "Var".IndTimerInicio := FALSE;
                   "Var".IndTimerTermino := FALSE;
                   "Var".Ind[2] := FALSE;
                   "Var".Ind[3] := FALSE;
                   "Var".Ind[4] := FALSE;
                   "Var".Ind[5] := FALSE;
                   "Var".Ind[6] := FALSE;
                   "Var".Ind[7] := FALSE;
                   "Var".Ind[8] := FALSE;
                   "Var".Ind[9] := FALSE;
                   "Var".Ind[10] := FALSE;
                   "Var".Ind[11] := FALSE;
               END_IF;

           END_REGION ;
           *)
       END_IF;

   END_IF;
END_REGION

REGION Network 5 (SCL): Puertas

   IF "Var".ActivarPuertaGA = TRUE THEN
       IF "Var".PuertaIniciada = FALSE AND "Var".PuertaInterrBounce = FALSE THEN
           "Var".PuertaIniciada := TRUE;
           "Var".PuertaInterrBounce := TRUE;
       END_IF;
       IF "Var".PuertaCerrando = TRUE AND ("lightBGround" = FALSE OR "lightB1" = FALSE OR "lightB2" = FALSE OR "lightB3" = FALSE) THEN
           "Var".PuertaInterrumpida := TRUE;
       END_IF;
       IF "Var".PuertaCerrando = TRUE AND "Var".PuertaInterrumpida = TRUE THEN
           "closeDoorG" := FALSE;
           "Var".PuertaCerrando := FALSE;
           "Var".PuertaInterrumpida := FALSE;
           "Var".PuertaAbriendo := TRUE;
           "Var".PuertaTimerTermino := FALSE;
           "openDoorG" := TRUE;
       END_IF;
       IF "Var".PuertaIniciada = TRUE AND "Var".PuertaAbriendo = FALSE AND "Var".PuertaAbierta = FALSE AND "Var".PuertaCerrando = FALSE AND "Var".PuertaTerminada = FALSE THEN
           IF "doorClosedG" = TRUE THEN
               "closeDoorG" := FALSE;
               "openDoorG" := TRUE;
               "Var".PuertaIniciada := FALSE;
               "Var".PuertaAbriendo := TRUE;
               "Var".PuertaTimerTermino := FALSE;
           END_IF;
       END_IF;
       IF "Var".PuertaIniciada = FALSE AND "Var".PuertaAbriendo = TRUE AND "Var".PuertaAbierta = FALSE AND "Var".PuertaCerrando = FALSE AND "Var".PuertaTerminada = FALSE THEN
           IF "doorOpenedG" = TRUE THEN
               "openDoorG" := FALSE;
               "Var".PuertaAbierta := TRUE;
               "Var".PuertaAbriendo := FALSE;
           END_IF;
       END_IF;
       IF "Var".PuertaIniciada = FALSE AND "Var".PuertaAbriendo = FALSE AND "Var".PuertaAbierta = TRUE AND "Var".PuertaCerrando = FALSE AND "Var".PuertaTerminada = FALSE THEN
           "Var".PuertaTimerInicio := TRUE;
           "Var".PuertaAbierta := FALSE;
       END_IF;
       "TimAbrir".TON(IN := "Var".PuertaTimerInicio,
                      PT := #TIMER,
                      Q  => "Var".PuertaTimerTermino);
       IF "Var".PuertaTimerTermino = TRUE THEN
           RESET_TIMER("TimAbrir");
           "closeDoorG" := TRUE;
           "Var".PuertaTimerTermino := FALSE;
           "Var".PuertaTimerInicio := FALSE;
           "Var".PuertaCerrando := TRUE;
       END_IF;
       IF "Var".PuertaIniciada = FALSE AND "Var".PuertaAbriendo = FALSE AND "Var".PuertaAbierta = FALSE AND "Var".PuertaCerrando = TRUE AND "Var".PuertaInterrumpida = FALSE AND "Var".PuertaTerminada = FALSE THEN
           IF "doorClosedG" = TRUE THEN
               "closeDoorG" := FALSE;
               "Var".PuertaCerrando := FALSE;
               "Var".PuertaTerminada := TRUE;
           END_IF;
       END_IF;
       IF "Var".PuertaIniciada = FALSE AND "Var".PuertaAbriendo = FALSE AND "Var".PuertaAbierta = FALSE AND "Var".PuertaCerrando = FALSE AND "Var".PuertaTerminada = TRUE THEN
           IF "doorClosedG" = TRUE AND "Var".PuertaTerminada = TRUE THEN
               "Var".PuertaTerminada := FALSE;
               "Var".PuertaInterrBounce := FALSE;
               "Var".ActivarPuertaGA := FALSE;
               "Var".ACCION := FALSE;
           END_IF;
       END_IF;
       IF "Var".PuertaIniciada = FALSE AND "Var".PuertaAbriendo = FALSE AND "Var".PuertaAbierta = FALSE AND "Var".PuertaCerrando = FALSE AND "Var".PuertaInterrumpida = FALSE AND "Var".PuertaTerminada = FALSE THEN
           "openDoorG" := FALSE;
           "closeDoorG" := FALSE;

       END_IF;
   END_IF;

   IF "Var".ActivarPuertaF1 = TRUE THEN
       IF "Var".PuertaIniciada = FALSE AND "Var".PuertaInterrBounce = FALSE THEN
           "Var".PuertaIniciada := TRUE;
           "Var".PuertaInterrBounce := TRUE;
       END_IF;
       IF "Var".PuertaCerrando = TRUE AND ("lightBGround" = FALSE OR "lightB1" = FALSE OR "lightB2" = FALSE OR "lightB3" = FALSE) THEN
           "Var".PuertaInterrumpida := TRUE;
       END_IF;
       IF "Var".PuertaCerrando = TRUE AND "Var".PuertaInterrumpida = TRUE THEN
           "closeDoor1" := FALSE;
           "Var".PuertaCerrando := FALSE;
           "Var".PuertaInterrumpida := FALSE;
           "Var".PuertaAbriendo := TRUE;
           "Var".PuertaTimerTermino := FALSE;
           "openDoor1" := TRUE;
       END_IF;
       IF "Var".PuertaIniciada = TRUE AND "Var".PuertaAbriendo = FALSE AND "Var".PuertaAbierta = FALSE AND "Var".PuertaCerrando = FALSE AND "Var".PuertaTerminada = FALSE THEN
           IF "doorClosed1" = TRUE THEN
               "closeDoor1" := FALSE;
               "openDoor1" := TRUE;
               "Var".PuertaIniciada := FALSE;
               "Var".PuertaAbriendo := TRUE;
               "Var".PuertaTimerTermino := FALSE;
           END_IF;
       END_IF;
       IF "Var".PuertaIniciada = FALSE AND "Var".PuertaAbriendo = TRUE AND "Var".PuertaAbierta = FALSE AND "Var".PuertaCerrando = FALSE AND "Var".PuertaTerminada = FALSE THEN
           IF "doorOpened1" = TRUE THEN
               "openDoor1" := FALSE;
               "Var".PuertaAbierta := TRUE;
               "Var".PuertaAbriendo := FALSE;
           END_IF;
       END_IF;
       IF "Var".PuertaIniciada = FALSE AND "Var".PuertaAbriendo = FALSE AND "Var".PuertaAbierta = TRUE AND "Var".PuertaCerrando = FALSE AND "Var".PuertaTerminada = FALSE THEN
           "Var".PuertaTimerInicio := TRUE;
           "Var".PuertaAbierta := FALSE;
       END_IF;
       "TimAbrir".TON(IN := "Var".PuertaTimerInicio,
                      PT := #TIMER,
                      Q  => "Var".PuertaTimerTermino);
       IF "Var".PuertaTimerTermino = TRUE THEN
           RESET_TIMER("TimAbrir");
           "closeDoor1" := TRUE;
           "Var".PuertaTimerTermino := FALSE;
           "Var".PuertaTimerInicio := FALSE;
           "Var".PuertaCerrando := TRUE;
       END_IF;
       IF "Var".PuertaIniciada = FALSE AND "Var".PuertaAbriendo = FALSE AND "Var".PuertaAbierta = FALSE AND "Var".PuertaCerrando = TRUE AND "Var".PuertaInterrumpida = FALSE AND "Var".PuertaTerminada = FALSE THEN
           IF "doorClosed1" = TRUE THEN
               "closeDoor1" := FALSE;
               "Var".PuertaCerrando := FALSE;
               "Var".PuertaTerminada := TRUE;
           END_IF;
       END_IF;
       IF "Var".PuertaIniciada = FALSE AND "Var".PuertaAbriendo = FALSE AND "Var".PuertaAbierta = FALSE AND "Var".PuertaCerrando = FALSE AND "Var".PuertaTerminada = TRUE THEN
           IF "doorClosed1" = TRUE AND "Var".PuertaTerminada = TRUE THEN
               "Var".PuertaTerminada := FALSE;
               "Var".PuertaInterrBounce := FALSE;
               "Var".ActivarPuertaF1 := FALSE;
               "Var".ACCION := FALSE;
           END_IF;
       END_IF;
       IF "Var".PuertaIniciada = FALSE AND "Var".PuertaAbriendo = FALSE AND "Var".PuertaAbierta = FALSE AND "Var".PuertaCerrando = FALSE AND "Var".PuertaInterrumpida = FALSE AND "Var".PuertaTerminada = FALSE THEN
           "openDoor1" := FALSE;
           "closeDoor1" := FALSE;

       END_IF;
   END_IF;

   IF "Var".ActivarPuertaF2 = TRUE THEN
       IF "Var".PuertaIniciada = FALSE AND "Var".PuertaInterrBounce = FALSE THEN
           "Var".PuertaIniciada := TRUE;
           "Var".PuertaInterrBounce := TRUE;
       END_IF;
       IF "Var".PuertaCerrando = TRUE AND ("lightBGround" = FALSE OR "lightB1" = FALSE OR "lightB2" = FALSE OR "lightB3" = FALSE) THEN
           "Var".PuertaInterrumpida := TRUE;
       END_IF;
       IF "Var".PuertaCerrando = TRUE AND "Var".PuertaInterrumpida = TRUE THEN
           "closeDoor2" := FALSE;
           "Var".PuertaCerrando := FALSE;
           "Var".PuertaInterrumpida := FALSE;
           "Var".PuertaAbriendo := TRUE;
           "Var".PuertaTimerTermino := FALSE;
           "openDoor2" := TRUE;
       END_IF;
       IF "Var".PuertaIniciada = TRUE AND "Var".PuertaAbriendo = FALSE AND "Var".PuertaAbierta = FALSE AND "Var".PuertaCerrando = FALSE AND "Var".PuertaTerminada = FALSE THEN
           IF "doorClosed2" = TRUE THEN
               "closeDoor2" := FALSE;
               "openDoor2" := TRUE;
               "Var".PuertaIniciada := FALSE;
               "Var".PuertaAbriendo := TRUE;
               "Var".PuertaTimerTermino := FALSE;
           END_IF;
       END_IF;
       IF "Var".PuertaIniciada = FALSE AND "Var".PuertaAbriendo = TRUE AND "Var".PuertaAbierta = FALSE AND "Var".PuertaCerrando = FALSE AND "Var".PuertaTerminada = FALSE THEN
           IF "doorOpened2" = TRUE THEN
               "openDoor2" := FALSE;
               "Var".PuertaAbierta := TRUE;
               "Var".PuertaAbriendo := FALSE;
           END_IF;
       END_IF;
       IF "Var".PuertaIniciada = FALSE AND "Var".PuertaAbriendo = FALSE AND "Var".PuertaAbierta = TRUE AND "Var".PuertaCerrando = FALSE AND "Var".PuertaTerminada = FALSE THEN
           "Var".PuertaTimerInicio := TRUE;
           "Var".PuertaAbierta := FALSE;
       END_IF;
       "TimAbrir".TON(IN := "Var".PuertaTimerInicio,
                      PT := #TIMER,
                      Q  => "Var".PuertaTimerTermino);
       IF "Var".PuertaTimerTermino = TRUE THEN
           RESET_TIMER("TimAbrir");
           "closeDoor2" := TRUE;
           "Var".PuertaTimerTermino := FALSE;
           "Var".PuertaTimerInicio := FALSE;
           "Var".PuertaCerrando := TRUE;
       END_IF;
       IF "Var".PuertaIniciada = FALSE AND "Var".PuertaAbriendo = FALSE AND "Var".PuertaAbierta = FALSE AND "Var".PuertaCerrando = TRUE AND "Var".PuertaInterrumpida = FALSE AND "Var".PuertaTerminada = FALSE THEN
           IF "doorClosed2" = TRUE THEN
               "closeDoor2" := FALSE;
               "Var".PuertaCerrando := FALSE;
               "Var".PuertaTerminada := TRUE;
           END_IF;
       END_IF;
       IF "Var".PuertaIniciada = FALSE AND "Var".PuertaAbriendo = FALSE AND "Var".PuertaAbierta = FALSE AND "Var".PuertaCerrando = FALSE AND "Var".PuertaTerminada = TRUE THEN
           IF "doorClosed2" = TRUE AND "Var".PuertaTerminada = TRUE THEN
               "Var".PuertaTerminada := FALSE;
               "Var".PuertaInterrBounce := FALSE;
               "Var".ActivarPuertaF2 := FALSE;
               "Var".ACCION := FALSE;
           END_IF;
       END_IF;
       IF "Var".PuertaIniciada = FALSE AND "Var".PuertaAbriendo = FALSE AND "Var".PuertaAbierta = FALSE AND "Var".PuertaCerrando = FALSE AND "Var".PuertaInterrumpida = FALSE AND "Var".PuertaTerminada = FALSE THEN
           "openDoor2" := FALSE;
           "closeDoor2" := FALSE;

       END_IF;
   END_IF;

   IF "Var".ActivarPuertaF3 = TRUE THEN
       IF "Var".PuertaIniciada = FALSE AND "Var".PuertaInterrBounce = FALSE THEN
           "Var".PuertaIniciada := TRUE;
           "Var".PuertaInterrBounce := TRUE;
       END_IF;
       IF "Var".PuertaCerrando = TRUE AND ("lightBGround" = FALSE OR "lightB1" = FALSE OR "lightB2" = FALSE OR "lightB3" = FALSE) THEN
           "Var".PuertaInterrumpida := TRUE;
       END_IF;
       IF "Var".PuertaCerrando = TRUE AND "Var".PuertaInterrumpida = TRUE THEN
           "closeDoor3" := FALSE;
           "Var".PuertaCerrando := FALSE;
           "Var".PuertaInterrumpida := FALSE;
           "Var".PuertaAbriendo := TRUE;
           "Var".PuertaTimerTermino := FALSE;
           "openDoor3" := TRUE;
       END_IF;
       IF "Var".PuertaIniciada = TRUE AND "Var".PuertaAbriendo = FALSE AND "Var".PuertaAbierta = FALSE AND "Var".PuertaCerrando = FALSE AND "Var".PuertaTerminada = FALSE THEN
           IF "doorClosed3" = TRUE THEN
               "closeDoor3" := FALSE;
               "openDoor3" := TRUE;
               "Var".PuertaIniciada := FALSE;
               "Var".PuertaAbriendo := TRUE;
               "Var".PuertaTimerTermino := FALSE;
           END_IF;
       END_IF;
       IF "Var".PuertaIniciada = FALSE AND "Var".PuertaAbriendo = TRUE AND "Var".PuertaAbierta = FALSE AND "Var".PuertaCerrando = FALSE AND "Var".PuertaTerminada = FALSE THEN
           IF "doorOpened3" = TRUE THEN
               "openDoor3" := FALSE;
               "Var".PuertaAbierta := TRUE;
               "Var".PuertaAbriendo := FALSE;
           END_IF;
       END_IF;
       IF "Var".PuertaIniciada = FALSE AND "Var".PuertaAbriendo = FALSE AND "Var".PuertaAbierta = TRUE AND "Var".PuertaCerrando = FALSE AND "Var".PuertaTerminada = FALSE THEN
           "Var".PuertaTimerInicio := TRUE;
           "Var".PuertaAbierta := FALSE;
       END_IF;
       "TimAbrir".TON(IN := "Var".PuertaTimerInicio,
                      PT := #TIMER,
                      Q  => "Var".PuertaTimerTermino);
       IF "Var".PuertaTimerTermino = TRUE THEN
           RESET_TIMER("TimAbrir");
           "closeDoor3" := TRUE;
           "Var".PuertaTimerTermino := FALSE;
           "Var".PuertaTimerInicio := FALSE;
           "Var".PuertaCerrando := TRUE;
       END_IF;
       IF "Var".PuertaIniciada = FALSE AND "Var".PuertaAbriendo = FALSE AND "Var".PuertaAbierta = FALSE AND "Var".PuertaCerrando = TRUE AND "Var".PuertaInterrumpida = FALSE AND "Var".PuertaTerminada = FALSE THEN
           IF "doorClosed3" = TRUE THEN
               "closeDoor3" := FALSE;
               "Var".PuertaCerrando := FALSE;
               "Var".PuertaTerminada := TRUE;
           END_IF;
       END_IF;
       IF "Var".PuertaIniciada = FALSE AND "Var".PuertaAbriendo = FALSE AND "Var".PuertaAbierta = FALSE AND "Var".PuertaCerrando = FALSE AND "Var".PuertaTerminada = TRUE THEN
           IF "doorClosed3" = TRUE AND "Var".PuertaTerminada = TRUE THEN
               "Var".PuertaTerminada := FALSE;
               "Var".PuertaInterrBounce := FALSE;
               "Var".ActivarPuertaF3 := FALSE;
               "Var".ACCION := FALSE;
           END_IF;
       END_IF;
       IF "Var".PuertaIniciada = FALSE AND "Var".PuertaAbriendo = FALSE AND "Var".PuertaAbierta = FALSE AND "Var".PuertaCerrando = FALSE AND "Var".PuertaInterrumpida = FALSE AND "Var".PuertaTerminada = FALSE THEN
           "openDoor3" := FALSE;
           "closeDoor3" := FALSE;

       END_IF;
   END_IF;
END_REGION

REGION Network 6 (SCL): Movimientos
   IF "Var".DeGAaF1 = TRUE THEN
       IF "Var".MovimientoLento = FALSE AND "Var".MovimientoRapido = FALSE AND "toZ+" = FALSE AND "toZ-" = FALSE THEN
           "Var".MovimientoLento := TRUE;
           "slow" := TRUE;
           "toZ+" := TRUE;
       END_IF;
       IF "Var".MovimientoLento = TRUE AND "Var".MovimientoRapido = FALSE AND "slowGround" = TRUE THEN
           "Var".MovimientoRapido := TRUE;
           "Var".MovimientoLento := FALSE;
           "slow" := FALSE;
       END_IF;
       IF "Var".MovimientoLento = FALSE AND "Var".MovimientoRapido = TRUE AND "slowBottom1" = TRUE THEN
           "Var".MovimientoRapido := FALSE;
           "Var".MovimientoLento := TRUE;
           "slow" := TRUE;
       END_IF;
       IF "Var".MovimientoLento = TRUE AND "Var".MovimientoRapido = FALSE AND "floorIndicator1" = TRUE THEN
           "Var".DeGAaF1 := FALSE;
           "Var".MovimientoRapido := FALSE;
           "Var".MovimientoLento := FALSE;
           "slow" := FALSE;
           "toZ+" := FALSE;
           "Var".Ind[3] := FALSE;
           "Var".Ind[4] := FALSE;
           "Var".Ind[9] := FALSE;
           "Var".ActivarPuertaF1 := TRUE;
       END_IF;
   END_IF;

   IF "Var".DeGAaF2 = TRUE THEN
       IF "Var".MovimientoLento = FALSE AND "Var".MovimientoRapido = FALSE AND "toZ+" = FALSE AND "toZ-" = FALSE THEN
           "Var".MovimientoLento := TRUE;
           "slow" := TRUE;
           "toZ+" := TRUE;
       END_IF;
       IF "Var".MovimientoLento = TRUE AND "Var".MovimientoRapido = FALSE AND "slowGround" = TRUE THEN
           "Var".MovimientoRapido := TRUE;
           "Var".MovimientoLento := FALSE;
           "slow" := FALSE;
       END_IF;
       IF "Var".MovimientoLento = FALSE AND "Var".MovimientoRapido = TRUE AND "slowBottom2" = TRUE THEN
           "Var".MovimientoRapido := FALSE;
           "Var".MovimientoLento := TRUE;
           "slow" := TRUE;
       END_IF;
       IF "Var".MovimientoLento = TRUE AND "Var".MovimientoRapido = FALSE AND "floorIndicator2" = TRUE THEN
           "Var".DeGAaF2 := FALSE;
           "Var".MovimientoRapido := FALSE;
           "Var".MovimientoLento := FALSE;
           "slow" := FALSE;
           "toZ+" := FALSE;
           "Var".Ind[5] := FALSE;
           "Var".Ind[6] := FALSE;
           "Var".Ind[10] := FALSE;
           "Var".ActivarPuertaF2 := TRUE;
       END_IF;
   END_IF;

   IF "Var".DeGAaF3 = TRUE THEN
       IF "Var".MovimientoLento = FALSE AND "Var".MovimientoRapido = FALSE AND "toZ+" = FALSE AND "toZ-" = FALSE THEN
           "Var".MovimientoLento := TRUE;
           "slow" := TRUE;
           "toZ+" := TRUE;
       END_IF;
       IF "Var".MovimientoLento = TRUE AND "Var".MovimientoRapido = FALSE AND "slowGround" = TRUE THEN
           "Var".MovimientoRapido := TRUE;
           "Var".MovimientoLento := FALSE;
           "slow" := FALSE;
       END_IF;
       IF "Var".MovimientoLento = FALSE AND "Var".MovimientoRapido = TRUE AND "slow3" = TRUE THEN
           "Var".MovimientoRapido := FALSE;
           "Var".MovimientoLento := TRUE;
           "slow" := TRUE;
       END_IF;
       IF "Var".MovimientoLento = TRUE AND "Var".MovimientoRapido = FALSE AND "floorIndicator3" = TRUE THEN
           "Var".DeGAaF3 := FALSE;
           "Var".MovimientoRapido := FALSE;
           "Var".MovimientoLento := FALSE;
           "slow" := FALSE;
           "toZ+" := FALSE;
           "Var".Ind[7] := FALSE;
           "Var".Ind[11] := FALSE;
           "Var".ActivarPuertaF3 := TRUE;
       END_IF;
   END_IF;

   IF "Var".DeF1aGA = TRUE THEN
       IF "Var".MovimientoLento = FALSE AND "Var".MovimientoRapido = FALSE AND "toZ+" = FALSE AND "toZ-" = FALSE THEN
           "Var".MovimientoLento := TRUE;
           "slow" := TRUE;
           "toZ-" := TRUE;
       END_IF;
       IF "Var".MovimientoLento = TRUE AND "Var".MovimientoRapido = FALSE AND "slowBottom1" = TRUE THEN
           "Var".MovimientoRapido := TRUE;
           "Var".MovimientoLento := FALSE;
           "slow" := FALSE;
       END_IF;
       IF "Var".MovimientoLento = FALSE AND "Var".MovimientoRapido = TRUE AND "slowGround" = TRUE THEN
           "Var".MovimientoRapido := FALSE;
           "Var".MovimientoLento := TRUE;
           "slow" := TRUE;
       END_IF;
       IF "Var".MovimientoLento = TRUE AND "Var".MovimientoRapido = FALSE AND "floorIndicatorG" = TRUE THEN
           "Var".DeF1aGA := FALSE;
           "Var".MovimientoRapido := FALSE;
           "Var".MovimientoLento := FALSE;
           "slow" := FALSE;
           "toZ-" := FALSE;
           "Var".Ind[2] := FALSE;
           "Var".Ind[8] := FALSE;
           "Var".ActivarPuertaGA := TRUE;
       END_IF;
   END_IF;

   IF "Var".DeF1aF2 = TRUE THEN
       IF "Var".MovimientoLento = FALSE AND "Var".MovimientoRapido = FALSE AND "toZ+" = FALSE AND "toZ-" = FALSE THEN
           "Var".MovimientoLento := TRUE;
           "slow" := TRUE;
           "toZ+" := TRUE;
       END_IF;
       IF "Var".MovimientoLento = TRUE AND "Var".MovimientoRapido = FALSE AND "slowTop1" = TRUE THEN
           "Var".MovimientoRapido := TRUE;
           "Var".MovimientoLento := FALSE;
           "slow" := FALSE;
       END_IF;
       IF "Var".MovimientoLento = FALSE AND "Var".MovimientoRapido = TRUE AND "slowBottom2" = TRUE THEN
           "Var".MovimientoRapido := FALSE;
           "Var".MovimientoLento := TRUE;
           "slow" := TRUE;
       END_IF;
       IF "Var".MovimientoLento = TRUE AND "Var".MovimientoRapido = FALSE AND "floorIndicator2" = TRUE THEN
           "Var".DeF1aF2 := FALSE;
           "Var".MovimientoRapido := FALSE;
           "Var".MovimientoLento := FALSE;
           "slow" := FALSE;
           "toZ+" := FALSE;
           "Var".Ind[5] := FALSE;
           "Var".Ind[6] := FALSE;
           "Var".Ind[10] := FALSE;
           "Var".ActivarPuertaF2 := TRUE;
       END_IF;
   END_IF;

   IF "Var".DeF1aF3 = TRUE THEN
       IF "Var".MovimientoLento = FALSE AND "Var".MovimientoRapido = FALSE AND "toZ+" = FALSE AND "toZ-" = FALSE THEN
           "Var".MovimientoLento := TRUE;
           "slow" := TRUE;
           "toZ+" := TRUE;
       END_IF;
       IF "Var".MovimientoLento = TRUE AND "Var".MovimientoRapido = FALSE AND "slowTop1" = TRUE THEN
           "Var".MovimientoRapido := TRUE;
           "Var".MovimientoLento := FALSE;
           "slow" := FALSE;
       END_IF;
       IF "Var".MovimientoLento = FALSE AND "Var".MovimientoRapido = TRUE AND "slow3" = TRUE THEN
           "Var".MovimientoRapido := FALSE;
           "Var".MovimientoLento := TRUE;
           "slow" := TRUE;
       END_IF;
       IF "Var".MovimientoLento = TRUE AND "Var".MovimientoRapido = FALSE AND "floorIndicator3" = TRUE THEN
           "Var".DeF1aF3 := FALSE;
           "Var".MovimientoRapido := FALSE;
           "Var".MovimientoLento := FALSE;
           "slow" := FALSE;
           "toZ+" := FALSE;
           "Var".Ind[7] := FALSE;
           "Var".Ind[11] := FALSE;
           "Var".ActivarPuertaF3 := TRUE;
       END_IF;
   END_IF;

   IF "Var".DeF2aGA = TRUE THEN
       IF "Var".MovimientoLento = FALSE AND "Var".MovimientoRapido = FALSE AND "toZ+" = FALSE AND "toZ-" = FALSE THEN
           "Var".MovimientoLento := TRUE;
           "slow" := TRUE;
           "toZ-" := TRUE;
       END_IF;
       IF "Var".MovimientoLento = TRUE AND "Var".MovimientoRapido = FALSE AND "slowBottom2" = TRUE THEN
           "Var".MovimientoRapido := TRUE;
           "Var".MovimientoLento := FALSE;
           "slow" := FALSE;
       END_IF;
       IF "Var".MovimientoLento = FALSE AND "Var".MovimientoRapido = TRUE AND "slowGround" = TRUE THEN
           "Var".MovimientoRapido := FALSE;
           "Var".MovimientoLento := TRUE;
           "slow" := TRUE;
       END_IF;
       IF "Var".MovimientoLento = TRUE AND "Var".MovimientoRapido = FALSE AND "floorIndicatorG" = TRUE THEN
           "Var".DeF2aGA := FALSE;
           "Var".MovimientoRapido := FALSE;
           "Var".MovimientoLento := FALSE;
           "slow" := FALSE;
           "toZ-" := FALSE;
           "Var".Ind[2] := FALSE;
           "Var".Ind[8] := FALSE;
           "Var".ActivarPuertaGA := TRUE;
       END_IF;
   END_IF;

   IF "Var".DeF2aF1 = TRUE THEN
       IF "Var".MovimientoLento = FALSE AND "Var".MovimientoRapido = FALSE AND "toZ+" = FALSE AND "toZ-" = FALSE THEN
           "Var".MovimientoLento := TRUE;
           "slow" := TRUE;
           "toZ-" := TRUE;
       END_IF;
       IF "Var".MovimientoLento = TRUE AND "Var".MovimientoRapido = FALSE AND "slowBottom2" = TRUE THEN
           "Var".MovimientoRapido := TRUE;
           "Var".MovimientoLento := FALSE;
           "slow" := FALSE;
       END_IF;
       IF "Var".MovimientoLento = FALSE AND "Var".MovimientoRapido = TRUE AND "slowTop1" = TRUE THEN
           "Var".MovimientoRapido := FALSE;
           "Var".MovimientoLento := TRUE;
           "slow" := TRUE;
       END_IF;
       IF "Var".MovimientoLento = TRUE AND "Var".MovimientoRapido = FALSE AND "floorIndicator1" = TRUE THEN
           "Var".DeF2aF1 := FALSE;
           "Var".MovimientoRapido := FALSE;
           "Var".MovimientoLento := FALSE;
           "slow" := FALSE;
           "toZ-" := FALSE;
           "Var".Ind[3] := FALSE;
           "Var".Ind[4] := FALSE;
           "Var".Ind[9] := FALSE;
           "Var".ActivarPuertaF1 := TRUE;
       END_IF;
   END_IF;

   IF "Var".DeF2aF3 = TRUE THEN
       IF "Var".MovimientoLento = FALSE AND "Var".MovimientoRapido = FALSE AND "toZ+" = FALSE AND "toZ-" = FALSE THEN
           "Var".MovimientoLento := TRUE;
           "slow" := TRUE;
           "toZ+" := TRUE;
       END_IF;
       IF "Var".MovimientoLento = TRUE AND "Var".MovimientoRapido = FALSE AND "slowTop2" = TRUE THEN
           "Var".MovimientoRapido := TRUE;
           "Var".MovimientoLento := FALSE;
           "slow" := FALSE;
       END_IF;
       IF "Var".MovimientoLento = FALSE AND "Var".MovimientoRapido = TRUE AND "slow3" = TRUE THEN
           "Var".MovimientoRapido := FALSE;
           "Var".MovimientoLento := TRUE;
           "slow" := TRUE;
       END_IF;
       IF "Var".MovimientoLento = TRUE AND "Var".MovimientoRapido = FALSE AND "floorIndicator3" = TRUE THEN
           "Var".DeF2aF3 := FALSE;
           "Var".MovimientoRapido := FALSE;
           "Var".MovimientoLento := FALSE;
           "slow" := FALSE;
           "toZ+" := FALSE;
           "Var".Ind[7] := FALSE;
           "Var".Ind[11] := FALSE;
           "Var".ActivarPuertaF3 := TRUE;
       END_IF;
   END_IF;

   IF "Var".DeF3aGA = TRUE THEN
       IF "Var".MovimientoLento = FALSE AND "Var".MovimientoRapido = FALSE AND "toZ+" = FALSE AND "toZ-" = FALSE THEN
           "Var".MovimientoLento := TRUE;
           "slow" := TRUE;
           "toZ-" := TRUE;
       END_IF;
       IF "Var".MovimientoLento = TRUE AND "Var".MovimientoRapido = FALSE AND "slow3" = TRUE THEN
           "Var".MovimientoRapido := TRUE;
           "Var".MovimientoLento := FALSE;
           "slow" := FALSE;
       END_IF;
       IF "Var".MovimientoLento = FALSE AND "Var".MovimientoRapido = TRUE AND "slowGround" = TRUE THEN
           "Var".MovimientoRapido := FALSE;
           "Var".MovimientoLento := TRUE;
           "slow" := TRUE;
       END_IF;
       IF "Var".MovimientoLento = TRUE AND "Var".MovimientoRapido = FALSE AND "floorIndicatorG" = TRUE THEN
           "Var".DeF3aGA := FALSE;
           "Var".MovimientoRapido := FALSE;
           "Var".MovimientoLento := FALSE;
           "slow" := FALSE;
           "toZ-" := FALSE;
           "Var".Ind[2] := FALSE;
           "Var".Ind[8] := FALSE;
           "Var".ActivarPuertaGA := TRUE;
       END_IF;
   END_IF;

   IF "Var".DeF3aF1 = TRUE THEN
       IF "Var".MovimientoLento = FALSE AND "Var".MovimientoRapido = FALSE AND "toZ+" = FALSE AND "toZ-" = FALSE THEN
           "Var".MovimientoLento := TRUE;
           "slow" := TRUE;
           "toZ-" := TRUE;
       END_IF;
       IF "Var".MovimientoLento = TRUE AND "Var".MovimientoRapido = FALSE AND "slow3" = TRUE THEN
           "Var".MovimientoRapido := TRUE;
           "Var".MovimientoLento := FALSE;
           "slow" := FALSE;
       END_IF;
       IF "Var".MovimientoLento = FALSE AND "Var".MovimientoRapido = TRUE AND "slowTop1" = TRUE THEN
           "Var".MovimientoRapido := FALSE;
           "Var".MovimientoLento := TRUE;
           "slow" := TRUE;
       END_IF;
       IF "Var".MovimientoLento = TRUE AND "Var".MovimientoRapido = FALSE AND "floorIndicator1" = TRUE THEN
           "Var".DeF3aF1 := FALSE;
           "Var".MovimientoRapido := FALSE;
           "Var".MovimientoLento := FALSE;
           "slow" := FALSE;
           "toZ-" := FALSE;
           "Var".Ind[3] := FALSE;
           "Var".Ind[4] := FALSE;
           "Var".Ind[9] := FALSE;
           "Var".ActivarPuertaF1 := TRUE;
       END_IF;
   END_IF;

   IF "Var".DeF3aF2 = TRUE THEN
       IF "Var".MovimientoLento = FALSE AND "Var".MovimientoRapido = FALSE AND "toZ+" = FALSE AND "toZ-" = FALSE THEN
           "Var".MovimientoLento := TRUE;
           "slow" := TRUE;
           "toZ-" := TRUE;
       END_IF;
       IF "Var".MovimientoLento = TRUE AND "Var".MovimientoRapido = FALSE AND "slow3" = TRUE THEN
           "Var".MovimientoRapido := TRUE;
           "Var".MovimientoLento := FALSE;
           "slow" := FALSE;
       END_IF;
       IF "Var".MovimientoLento = FALSE AND "Var".MovimientoRapido = TRUE AND "slowTop2" = TRUE THEN
           "Var".MovimientoRapido := FALSE;
           "Var".MovimientoLento := TRUE;
           "slow" := TRUE;
       END_IF;
       IF "Var".MovimientoLento = TRUE AND "Var".MovimientoRapido = FALSE AND "floorIndicator2" = TRUE THEN
           "Var".DeF3aF2 := FALSE;
           "Var".MovimientoRapido := FALSE;
           "Var".MovimientoLento := FALSE;
           "slow" := FALSE;
           "toZ-" := FALSE;
           "Var".Ind[5] := FALSE;
           "Var".Ind[6] := FALSE;
           "Var".Ind[10] := FALSE;
           "Var".ActivarPuertaF2 := TRUE;
       END_IF;
   END_IF;
END_REGION

REGION Network 7 (SCL): Simulador Estados
   IF "posGround" = TRUE AND "doorClosedG" THEN
       "Var".SimuladorEstado1 := TRUE;
       "Var".SimuladorEstado2 := FALSE;
       "Var".SimuladorEstado3 := FALSE;
       "Var".SimuladorEstado4 := FALSE;
       "Var".SimuladorEstado5 := FALSE;
       "Var".SimuladorEstado6 := FALSE;
       "Var".SimuladorEstado7 := FALSE;
       "Var".SimuladorEstado8 := FALSE;
   END_IF;

   IF "posGround" = TRUE AND "doorOpenedG" THEN
       "Var".SimuladorEstado1 := FALSE;
       "Var".SimuladorEstado2 := TRUE;
       "Var".SimuladorEstado3 := FALSE;
       "Var".SimuladorEstado4 := FALSE;
       "Var".SimuladorEstado5 := FALSE;
       "Var".SimuladorEstado6 := FALSE;
       "Var".SimuladorEstado7 := FALSE;
       "Var".SimuladorEstado8 := FALSE;
   END_IF;

   IF "posFloor1" = TRUE AND "doorClosed1" THEN
       "Var".SimuladorEstado1 := FALSE;
       "Var".SimuladorEstado2 := FALSE;
       "Var".SimuladorEstado3 := TRUE;
       "Var".SimuladorEstado4 := FALSE;
       "Var".SimuladorEstado5 := FALSE;
       "Var".SimuladorEstado6 := FALSE;
       "Var".SimuladorEstado7 := FALSE;
       "Var".SimuladorEstado8 := FALSE;
   END_IF;

   IF "posFloor1" = TRUE AND "doorOpened1" THEN
       "Var".SimuladorEstado1 := FALSE;
       "Var".SimuladorEstado2 := FALSE;
       "Var".SimuladorEstado3 := FALSE;
       "Var".SimuladorEstado4 := TRUE;
       "Var".SimuladorEstado5 := FALSE;
       "Var".SimuladorEstado6 := FALSE;
       "Var".SimuladorEstado7 := FALSE;
       "Var".SimuladorEstado8 := FALSE;
   END_IF;

   IF "posFloor2" = TRUE AND "doorClosed2" THEN
       "Var".SimuladorEstado1 := FALSE;
       "Var".SimuladorEstado2 := FALSE;
       "Var".SimuladorEstado3 := FALSE;
       "Var".SimuladorEstado4 := FALSE;
       "Var".SimuladorEstado5 := TRUE;
       "Var".SimuladorEstado6 := FALSE;
       "Var".SimuladorEstado7 := FALSE;
       "Var".SimuladorEstado8 := FALSE;
   END_IF;

   IF "posFloor2" = TRUE AND "doorOpened2" THEN
       "Var".SimuladorEstado1 := FALSE;
       "Var".SimuladorEstado2 := FALSE;
       "Var".SimuladorEstado3 := FALSE;
       "Var".SimuladorEstado4 := FALSE;
       "Var".SimuladorEstado5 := FALSE;
       "Var".SimuladorEstado6 := TRUE;
       "Var".SimuladorEstado7 := FALSE;
       "Var".SimuladorEstado8 := FALSE;
   END_IF;

   IF "posFloor3" = TRUE AND "doorClosed3" THEN
       "Var".SimuladorEstado1 := FALSE;
       "Var".SimuladorEstado2 := FALSE;
       "Var".SimuladorEstado3 := FALSE;
       "Var".SimuladorEstado4 := FALSE;
       "Var".SimuladorEstado5 := FALSE;
       "Var".SimuladorEstado6 := FALSE;
       "Var".SimuladorEstado7 := TRUE;
       "Var".SimuladorEstado8 := FALSE;
   END_IF;

   IF "posFloor3" = TRUE AND "doorOpened3" THEN
       "Var".SimuladorEstado1 := FALSE;
       "Var".SimuladorEstado2 := FALSE;
       "Var".SimuladorEstado3 := FALSE;
       "Var".SimuladorEstado4 := FALSE;
       "Var".SimuladorEstado5 := FALSE;
       "Var".SimuladorEstado6 := FALSE;
       "Var".SimuladorEstado7 := FALSE;
       "Var".SimuladorEstado8 := TRUE;
   END_IF;
END_REGION

REGION Network 8 (SCL): Master Activado
   IF "Var".MasterBounceThree = FALSE AND "Var".MASTER = FALSE AND "Var".MasterBounceOne = FALSE AND "Var".MasterBounceTwo = FALSE THEN
       "Var".MASTERINDICATOR := FALSE;
   END_IF;
   IF "Var".MASTERINDICATOR = FALSE AND "Var".MASTER = TRUE AND "Var".MasterBounceOne = FALSE AND "Var".MasterBounceTwo = FALSE THEN
       "Var".MasterBounceThree := TRUE;
       "Var".MasterBounceOne := TRUE;
   END_IF;
   IF "Var".MasterBounceThree = TRUE AND "Var".MASTER = FALSE AND "Var".MasterBounceOne = TRUE THEN
       "Var".MASTERINDICATOR := TRUE;
       "Var".MasterBounceTwo := TRUE;
   END_IF;
   IF "Var".MasterBounceThree = TRUE AND "Var".MASTER = TRUE AND "Var".MasterBounceOne = TRUE AND "Var".MasterBounceTwo = TRUE THEN
       "Var".MasterBounceThree := FALSE;
   END_IF;
   IF "Var".MasterBounceThree = FALSE AND "Var".MASTER = FALSE AND "Var".MasterBounceOne = TRUE AND "Var".MasterBounceTwo = TRUE THEN
       "Var".MASTERINDICATOR := FALSE;
       "Var".MasterBounceOne := FALSE;
       "Var".MasterBounceTwo := FALSE;
       "Var".ResetApplied := FALSE;
       "Var".MasterResetPos := TRUE;
   END_IF;

   IF "Var".MasterResetPos = TRUE THEN
       IF "posGround" = FALSE THEN
           IF "Var".MovimientoRapido = FALSE AND "toZ+" = FALSE AND "toZ-" = FALSE AND "slow" = FALSE THEN
               "Var".MovimientoRapido := TRUE;
               "toZ-" := TRUE;
           END_IF;
           IF "Var".MovimientoRapido = TRUE AND "slowGround" = TRUE AND "slow" = FALSE THEN
               "Var".MovimientoRapido := FALSE;
               "slow" := TRUE;
           END_IF;
       END_IF;
       IF "posGround" = TRUE THEN
           "slow" := FALSE;
           "toZ-" := FALSE;
           "Var".MasterResetPos := FALSE;
           "Var".MasterResPosPuerta := TRUE;
       END_IF;
   END_IF;

   IF "Var".MasterResPosPuerta = TRUE THEN
       IF "doorClosedG" = TRUE AND "Var".MasterPuertaG = FALSE THEN
           "closeDoorG" := FALSE;
           "openDoorG" := FALSE;
       END_IF;
       IF "doorClosedG" = TRUE AND "Var".MasterPuertaG = TRUE THEN
           "closeDoorG" := FALSE;
           "openDoorG" := FALSE;
           "Var".MasterPuerta1 := FALSE;
       END_IF;
       IF "doorClosedG" = FALSE AND "Var".MasterPuertaG = FALSE THEN
           "closeDoorG" := TRUE;
           "openDoorG" := FALSE;
           "Var".MasterPuertaG := TRUE;
       END_IF;

       IF "doorClosed1" = TRUE AND "Var".MasterPuerta1 = FALSE THEN
           "closeDoor1" := FALSE;
           "openDoor1" := FALSE;
       END_IF;
       IF "doorClosed1" = TRUE AND "Var".MasterPuerta1 = TRUE THEN
           "closeDoor1" := FALSE;
           "openDoor1" := FALSE;
           "Var".MasterPuerta1 := FALSE;
       END_IF;
       IF "doorClosed1" = FALSE AND "Var".MasterPuerta1 = FALSE THEN
           "closeDoor1" := TRUE;
           "openDoor1" := FALSE;
           "Var".MasterPuerta1 := TRUE;
       END_IF;

       IF "doorClosed2" = TRUE AND "Var".MasterPuerta2 = FALSE THEN
           "closeDoor2" := FALSE;
           "openDoor2" := FALSE;
       END_IF;
       IF "doorClosed2" = TRUE AND "Var".MasterPuerta2 = TRUE THEN
           "closeDoor2" := FALSE;
           "openDoor2" := FALSE;
           "Var".MasterPuerta2 := FALSE;
       END_IF;
       IF "doorClosed2" = FALSE AND "Var".MasterPuerta2 = FALSE THEN
           "closeDoor2" := TRUE;
           "openDoor2" := FALSE;
           "Var".MasterPuerta2 := TRUE;
       END_IF;

       IF "doorClosed3" = TRUE AND "Var".MasterPuerta3 = FALSE THEN
           "closeDoor3" := FALSE;
           "openDoor3" := FALSE;
       END_IF;
       IF "doorClosed3" = TRUE AND "Var".MasterPuerta3 = TRUE THEN
           "closeDoor3" := FALSE;
           "openDoor3" := FALSE;
           "Var".MasterPuerta3 := FALSE;
       END_IF;
       IF "doorClosed3" = FALSE AND "Var".MasterPuerta3 = FALSE THEN
           "closeDoor3" := TRUE;
           "openDoor3" := FALSE;
           "Var".MasterPuerta3 := TRUE;
       END_IF;

       IF "doorClosedG" = TRUE AND "doorClosed1" = TRUE AND "doorClosed2" = TRUE AND "doorClosed3" = TRUE THEN
           "Var".MasterResPosPuerta := FALSE;
       END_IF;

   END_IF;
END_REGION

REGION Network 9 (SCL): RESET
   IF "Var".RESET = TRUE THEN
       FOR #i := 0 TO 10 DO
           "Var".Acc[#i] := 'EMPTY';
           "Var".AccMovTemp[#i] := 'EMPTY';
       END_FOR;
       FILL_BLK(IN    := FALSE,
                COUNT := 15,
                OUT   => "Var".Ind[0]);
       FILL_BLK(IN    := FALSE,
                COUNT := 15,
                OUT   => "Var".AccSucc[0]);

       RESET_TIMER("TimAbrir");

       "Var".tempStringOne := '';
       "Var".tempStringTwo := '';
       "Var".bounceOneAlerta := FALSE;
       "Var".bounceTwoAlerta := FALSE;
       "Var".bounceOneEmergen := FALSE;
       "Var".bounceTwoEmergen := FALSE;
       "Var".bounceOneGroundA := FALSE;
       "Var".sendAccGroundA := FALSE;
       "Var".sendAccF1DownA := FALSE;
       "Var".PuertaIniciada := FALSE;
       "Var".PuertaAbriendo := FALSE;
       "Var".PuertaAbierta := FALSE;
       "Var".PuertaCerrando := FALSE;
       "Var".PuertaInterrumpida := FALSE;
       "Var".PuertaTerminada := FALSE;
       "Var".PuertaTimerInicio := FALSE;
       "Var".PuertaTimerTermino := FALSE;
       "Var".PuertaInterrBounce := FALSE;
       "Var".ActivarPuertaGA := FALSE;
       "Var".ActivarPuertaF1 := FALSE;
       "Var".ActivarPuertaF2 := FALSE;
       "Var".ActivarPuertaF3 := FALSE;
       "Var".bounceOneF1DownA := FALSE;
       "Var".sendAccF1DownA := FALSE;
       "Var".ACCION := FALSE;
       "Var".DeGAaF1 := FALSE;
       "Var".DeGAaF2 := FALSE;
       "Var".DeGAaF3 := FALSE;
       "Var".DeF1aGA := FALSE;
       "Var".DeF1aF2 := FALSE;
       "Var".DeF1aF3 := FALSE;
       "Var".DeF2aGA := FALSE;
       "Var".DeF2aF1 := FALSE;
       "Var".DeF2aF3 := FALSE;
       "Var".DeF3aGA := FALSE;
       "Var".DeF3aF1 := FALSE;
       "Var".DeF3aF2 := FALSE;
       "Var".MOVIMIENTO := FALSE;
       "Var".MovimientoLento := FALSE;
       "Var".MovimientoRapido := FALSE;
       "Var".SimuladorEstado1 := FALSE;
       "Var".SimuladorEstado2 := FALSE;
       "Var".SimuladorEstado3 := FALSE;
       "Var".SimuladorEstado4 := FALSE;
       "Var".SimuladorEstado5 := FALSE;
       "Var".SimuladorEstado6 := FALSE;
       "Var".SimuladorEstado7 := FALSE;
       "Var".SimuladorEstado8 := FALSE;
       "Var".MasterPuertaG := FALSE;
       "Var".MasterPuerta1 := FALSE;
       "Var".MasterPuerta2 := FALSE;
       "Var".MasterPuerta3 := FALSE;

       "toZ+" := FALSE;
       "toZ-" := FALSE;
       "slow" := FALSE;
       "openDoorG" := FALSE;
       "openDoor1" := FALSE;
       "openDoor2" := FALSE;
       "openDoor3" := FALSE;
       "closeDoorG" := FALSE;
       "closeDoor1" := FALSE;
       "closeDoor2" := FALSE;
       "closeDoor3" := FALSE;
       "callToGround" := FALSE;
       "callToDown1" := FALSE;
       "callToDown2" := FALSE;
       "callTo3" := FALSE;
       "sendToGround" := FALSE;
       "sendTo1" := FALSE;
       "sendTo2" := FALSE;
       "sendTo3" := FALSE;
       "alertInd" := FALSE;
       "emergencyInd" := FALSE;
       "overloadInd" := FALSE;
       "sendGroundMaster" := FALSE;
       "send1Master" := FALSE;
       "send2Master" := FALSE;
       "send3Master" := FALSE;
       "alertMaster" := FALSE;
       "emergencyMaster" := FALSE;
       "abrirPuertasMaster" := FALSE;
       "cerrarPuertasMaster" := FALSE;

       //Floor Indicator and CabinUpDown Nope

       "Var".RESET := FALSE;
   END_IF;
END_REGION

REGION Network 10 (SCL): Puertas Master

   IF "Var".MASTERINDICATOR = TRUE THEN

       //Abrir y cerrar puerta ground
       IF "posGround" = TRUE AND "doorClosedG" = FALSE AND "cerrarPuertasMaster" = TRUE AND "Var".MasterPuertaGBounce = FALSE AND "Var".MasterPuertaGBounce2 = FALSE THEN
           "Var".MasterPuertaGBounce := TRUE;
       END_IF;
       IF "tempFloor1" = TRUE AND "doorClosedG" = FALSE AND "cerrarPuertasMaster" = TRUE AND "Var".MasterPuertaGBounce = FALSE AND "Var".MasterPuertaGBounce2 = TRUE THEN
           "closeDoorG" := FALSE;
           "openDoorG" := FALSE;
           "Var".MasterPuertaGBounce := TRUE;
           "Var".MasterPuertaGBounce2 := FALSE;
       END_IF;
       IF "tempFloor1" = TRUE AND "doorClosedG" = FALSE AND "Var".MasterPuertaGBounce = TRUE THEN
           "closeDoorG" := TRUE;
           "openDoorG" := FALSE;
       END_IF;
       IF "tempFloor1" = TRUE AND "doorClosedG" = TRUE AND "Var".MasterPuertaGBounce = TRUE THEN
           "closeDoorG" := FALSE;
           "openDoorG" := FALSE;
           "Var".MasterPuertaGBounce := FALSE;
       END_IF;
       IF "posGround" = TRUE AND "doorOpenedG" = FALSE AND "abrirPuertasMaster" = TRUE AND "Var".MasterPuertaGBounce2 = FALSE AND "Var".MasterPuertaGBounce = FALSE THEN
           "Var".MasterPuertaGBounce2 := TRUE;
       END_IF;
       IF "tempFloor1" = TRUE AND "doorOpenedG" = FALSE AND "abrirPuertasMaster" = TRUE AND "Var".MasterPuertaGBounce2 = FALSE AND "Var".MasterPuertaGBounce = TRUE THEN
           "closeDoorG" := FALSE;
           "openDoorG" := FALSE;
           "Var".MasterPuertaGBounce := FALSE;
           "Var".MasterPuertaGBounce2 := TRUE;
       END_IF;
       IF "tempFloor1" = TRUE AND "doorOpenedG" = FALSE AND "Var".MasterPuertaGBounce2 = TRUE THEN
           "closeDoorG" := FALSE;
           "openDoorG" := TRUE;
       END_IF;
       IF "tempFloor1" = TRUE AND "doorOpenedG" = TRUE AND "Var".MasterPuertaGBounce2 = TRUE THEN
           "closeDoorG" := FALSE;
           "openDoorG" := FALSE;
           "Var".MasterPuertaGBounce := FALSE;
       END_IF;

       //Abrir y cerrar puerta floor 1
       IF "posFloor1" = TRUE AND "doorClosed1" = FALSE AND "cerrarPuertasMaster" = TRUE AND "Var".MasterPuerta1Bounce = FALSE AND "Var".MasterPuerta1Bounce2 = FALSE THEN
           "Var".MasterPuerta1Bounce := TRUE;
       END_IF;
       IF ("tempFloor2" = TRUE OR "tempFloor4" = TRUE) AND "doorClosed1" = FALSE AND "cerrarPuertasMaster" = TRUE AND "Var".MasterPuerta1Bounce = FALSE AND "Var".MasterPuerta1Bounce2 = TRUE THEN
           "closeDoor1" := FALSE;
           "openDoor1" := FALSE;
           "Var".MasterPuerta1Bounce := TRUE;
           "Var".MasterPuerta1Bounce2 := FALSE;
       END_IF;
       IF ("tempFloor2" = TRUE OR "tempFloor4" = TRUE) AND "doorClosed1" = FALSE AND "Var".MasterPuerta1Bounce = TRUE THEN
           "closeDoor1" := TRUE;
           "openDoor1" := FALSE;
       END_IF;
       IF ("tempFloor2" = TRUE OR "tempFloor4" = TRUE) AND "doorClosed1" = TRUE AND "Var".MasterPuerta1Bounce = TRUE THEN
           "closeDoor1" := FALSE;
           "openDoor1" := FALSE;
           "Var".MasterPuerta1Bounce := FALSE;
       END_IF;
       IF "posFloor1" = TRUE AND "doorOpened1" = FALSE AND "abrirPuertasMaster" = TRUE AND "Var".MasterPuerta1Bounce2 = FALSE AND "Var".MasterPuerta1Bounce = FALSE THEN
           "Var".MasterPuerta1Bounce2 := TRUE;
       END_IF;
       IF ("tempFloor2" = TRUE OR "tempFloor4" = TRUE) AND "doorOpened1" = FALSE AND "abrirPuertasMaster" = TRUE AND "Var".MasterPuerta1Bounce2 = FALSE AND "Var".MasterPuerta1Bounce = TRUE THEN
           "closeDoor1" := FALSE;
           "openDoor1" := FALSE;
           "Var".MasterPuerta1Bounce := FALSE;
           "Var".MasterPuerta1Bounce2 := TRUE;
       END_IF;
       IF ("tempFloor2" = TRUE OR "tempFloor4" = TRUE) AND "doorOpened1" = FALSE AND "Var".MasterPuerta1Bounce2 = TRUE THEN
           "closeDoor1" := FALSE;
           "openDoor1" := TRUE;
       END_IF;
       IF ("tempFloor2" = TRUE OR "tempFloor4" = TRUE) AND "doorOpened1" = TRUE AND "Var".MasterPuerta1Bounce2 = TRUE THEN
           "closeDoor1" := FALSE;
           "openDoor1" := FALSE;
           "Var".MasterPuerta1Bounce := FALSE;
       END_IF;

       //Abrir y cerrar puerta floor 2
       IF "posFloor2" = TRUE AND "doorClosed2" = FALSE AND "cerrarPuertasMaster" = TRUE AND "Var".MasterPuerta2Bounce = FALSE AND "Var".MasterPuerta2Bounce2 = FALSE THEN
           "Var".MasterPuerta2Bounce := TRUE;
       END_IF;
       IF ("tempFloor5" = TRUE OR "tempFloor7" = TRUE) AND "doorClosed2" = FALSE AND "cerrarPuertasMaster" = TRUE AND "Var".MasterPuerta2Bounce = FALSE AND "Var".MasterPuerta2Bounce2 = TRUE THEN
           "closeDoor2" := FALSE;
           "openDoor2" := FALSE;
           "Var".MasterPuerta2Bounce := TRUE;
           "Var".MasterPuerta2Bounce2 := FALSE;
       END_IF;
       IF ("tempFloor5" = TRUE OR "tempFloor7" = TRUE) AND "doorClosed2" = FALSE AND "Var".MasterPuerta2Bounce = TRUE THEN
           "closeDoor2" := TRUE;
           "openDoor2" := FALSE;
       END_IF;
       IF ("tempFloor5" = TRUE OR "tempFloor7" = TRUE) AND "doorClosed2" = TRUE AND "Var".MasterPuerta2Bounce = TRUE THEN
           "closeDoor2" := FALSE;
           "openDoor2" := FALSE;
           "Var".MasterPuerta2Bounce := FALSE;
       END_IF;
       IF "posFloor2" = TRUE AND "doorOpened2" = FALSE AND "abrirPuertasMaster" = TRUE AND "Var".MasterPuerta2Bounce2 = FALSE AND "Var".MasterPuerta2Bounce = FALSE THEN
           "Var".MasterPuerta2Bounce2 := TRUE;
       END_IF;
       IF ("tempFloor5" = TRUE OR "tempFloor7" = TRUE) AND "doorOpened2" = FALSE AND "abrirPuertasMaster" = TRUE AND "Var".MasterPuerta2Bounce2 = FALSE AND "Var".MasterPuerta2Bounce = TRUE THEN
           "closeDoor2" := FALSE;
           "openDoor2" := FALSE;
           "Var".MasterPuerta2Bounce := FALSE;
           "Var".MasterPuerta2Bounce2 := TRUE;
       END_IF;
       IF ("tempFloor5" = TRUE OR "tempFloor7" = TRUE) AND "doorOpened2" = FALSE AND "Var".MasterPuerta2Bounce2 = TRUE THEN
           "closeDoor2" := FALSE;
           "openDoor2" := TRUE;
       END_IF;
       IF ("tempFloor5" = TRUE OR "tempFloor7" = TRUE) AND "doorOpened2" = TRUE AND "Var".MasterPuerta2Bounce2 = TRUE THEN
           "closeDoor2" := FALSE;
           "openDoor2" := FALSE;
           "Var".MasterPuerta2Bounce := FALSE;
       END_IF;

       //Abrir y cerrar puerta floor 3
       IF "posFloor3" = TRUE AND "doorClosed3" = FALSE AND "cerrarPuertasMaster" = TRUE AND "Var".MasterPuerta3Bounce = FALSE AND "Var".MasterPuerta3Bounce2 = FALSE THEN
           "Var".MasterPuerta3Bounce := TRUE;
       END_IF;
       IF "tempFloor6" = TRUE AND "doorClosed3" = FALSE AND "cerrarPuertasMaster" = TRUE AND "Var".MasterPuerta3Bounce = FALSE AND "Var".MasterPuerta3Bounce2 = TRUE THEN
           "closeDoor3" := FALSE;
           "openDoor3" := FALSE;
           "Var".MasterPuerta3Bounce := TRUE;
           "Var".MasterPuerta3Bounce2 := FALSE;
       END_IF;
       IF "tempFloor6" = TRUE AND "doorClosed3" = FALSE AND "Var".MasterPuerta3Bounce = TRUE THEN
           "closeDoor3" := TRUE;
           "openDoor3" := FALSE;
       END_IF;
       IF "tempFloor6" = TRUE AND "doorClosed3" = TRUE AND "Var".MasterPuerta3Bounce = TRUE THEN
           "closeDoor3" := FALSE;
           "openDoor3" := FALSE;
           "Var".MasterPuerta3Bounce := FALSE;
       END_IF;
       IF "posFloor3" = TRUE AND "doorOpened3" = FALSE AND "abrirPuertasMaster" = TRUE AND "Var".MasterPuerta3Bounce2 = FALSE AND "Var".MasterPuerta3Bounce = FALSE THEN
           "Var".MasterPuerta3Bounce2 := TRUE;
       END_IF;
       IF "tempFloor6" = TRUE AND "doorOpened3" = FALSE AND "abrirPuertasMaster" = TRUE AND "Var".MasterPuerta3Bounce2 = FALSE AND "Var".MasterPuerta3Bounce = TRUE THEN
           "closeDoor3" := FALSE;
           "openDoor3" := FALSE;
           "Var".MasterPuerta3Bounce := FALSE;
           "Var".MasterPuerta3Bounce2 := TRUE;
       END_IF;
       IF "tempFloor6" = TRUE AND "doorOpened3" = FALSE AND "Var".MasterPuerta3Bounce2 = TRUE THEN
           "closeDoor3" := FALSE;
           "openDoor3" := TRUE;
       END_IF;
       IF "tempFloor6" = TRUE AND "doorOpened3" = TRUE AND "Var".MasterPuerta3Bounce2 = TRUE THEN
           "closeDoor3" := FALSE;
           "openDoor3" := FALSE;
           "Var".MasterPuerta3Bounce := FALSE;
       END_IF;

   END_IF;
END_REGION

REGION Network 11 (SCL): Movimientos Master
   //Se quito encendido y direccion del movimiento si no ha llegado al otro
   IF "Var".MASTERINDICATOR = TRUE THEN

       //Ir a Ground
       IF "posGround" = FALSE AND "sendGroundMaster" = TRUE AND "Var".MasterSendToGround = FALSE THEN
           "slow" := FALSE;
           "toZ-" := FALSE;
           "toZ+" := FALSE;
           "Var".MasterSendToGroundB2 := FALSE;
           "Var".MasterSendToGroundB := FALSE;
           "Var".MasterSendToGround := TRUE;
           "Var".MasterSendTo1 := FALSE;
           "Var".MasterSendTo1B := FALSE;
           "Var".MasterSendTo1B2 := FALSE;
           "Var".MasterSendTo2 := FALSE;
           "Var".MasterSendTo2B := FALSE;
           "Var".MasterSendTo2B2 := FALSE;
           "Var".MasterSendTo3 := FALSE;
           "Var".MasterSendTo3B := FALSE;
           "Var".MasterSendTo3B2 := FALSE;
           "sendToGroundMaster" := FALSE;
           "sendTo1Master" := FALSE;
           "sendTo2Master" := FALSE;
           "sendTo3Master" := FALSE;
       END_IF;
       IF "Var".MasterSendToGround = TRUE THEN
           IF "Var".MasterSendToGroundB = FALSE THEN
               "Var".MasterSendToGroundB := TRUE;
               "toZ-" := TRUE;
               "sendToGroundMaster" := TRUE;
           END_IF;
           IF "Var".MasterSendToGroundB = TRUE AND "toZ-" = TRUE AND "slowGround" = TRUE AND "slow" = FALSE THEN
               "Var".MasterSendToGroundB := FALSE;
               "Var".MasterSendToGroundB2 := TRUE;
               "slow" := TRUE;
           END_IF;
           IF "posGround" = TRUE  THEN
               "slow" := FALSE;
               "toZ-" := FALSE;
               "Var".MasterSendToGroundB2 := FALSE;
               "Var".MasterSendToGroundB := FALSE;
               "Var".MasterSendToGround := FALSE;
               "sendToGroundMaster" := FALSE;
           END_IF;
       END_IF;

